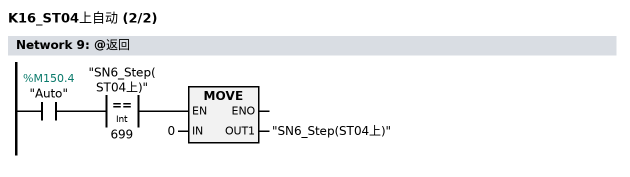
   RUNG wire#powerrail
      Contact( "Auto" )
      { S7_Templates := "SrcType := Int" } EQ_Contact(in1 := "SN6_Step(ST04上)", in2 := 699)
      Move(in := 0, out1 => "SN6_Step(ST04上)")
   END_RUNG
   // the same network as SCL:
   IF "Auto" AND ("SN6_Step(ST04上)" = 699) THEN "SN6_Step(ST04上)" := 0; END_IF;
END_REGION
END_FUNCTION_BLOCK

FUNCTION_BLOCK "K17_ST05上自动"   // FB17, LAD
{ S7_Optimized_Access := 'TRUE' }
VERSION : 0.1
// stored: AutoNumber false, IsIECCheckEnabled false, IsRetainMemResEnabled false, MemoryReserve 100, SetENOAutomatically false, UDAEnableTagReadback false
   VAR_TEMP   // added for the SCL form of the ladder/FBD networks
      _w1 : Bool;
   END_VAR
BEGIN

REGION Network 2: @搬出条件，SN7===ST05上工位
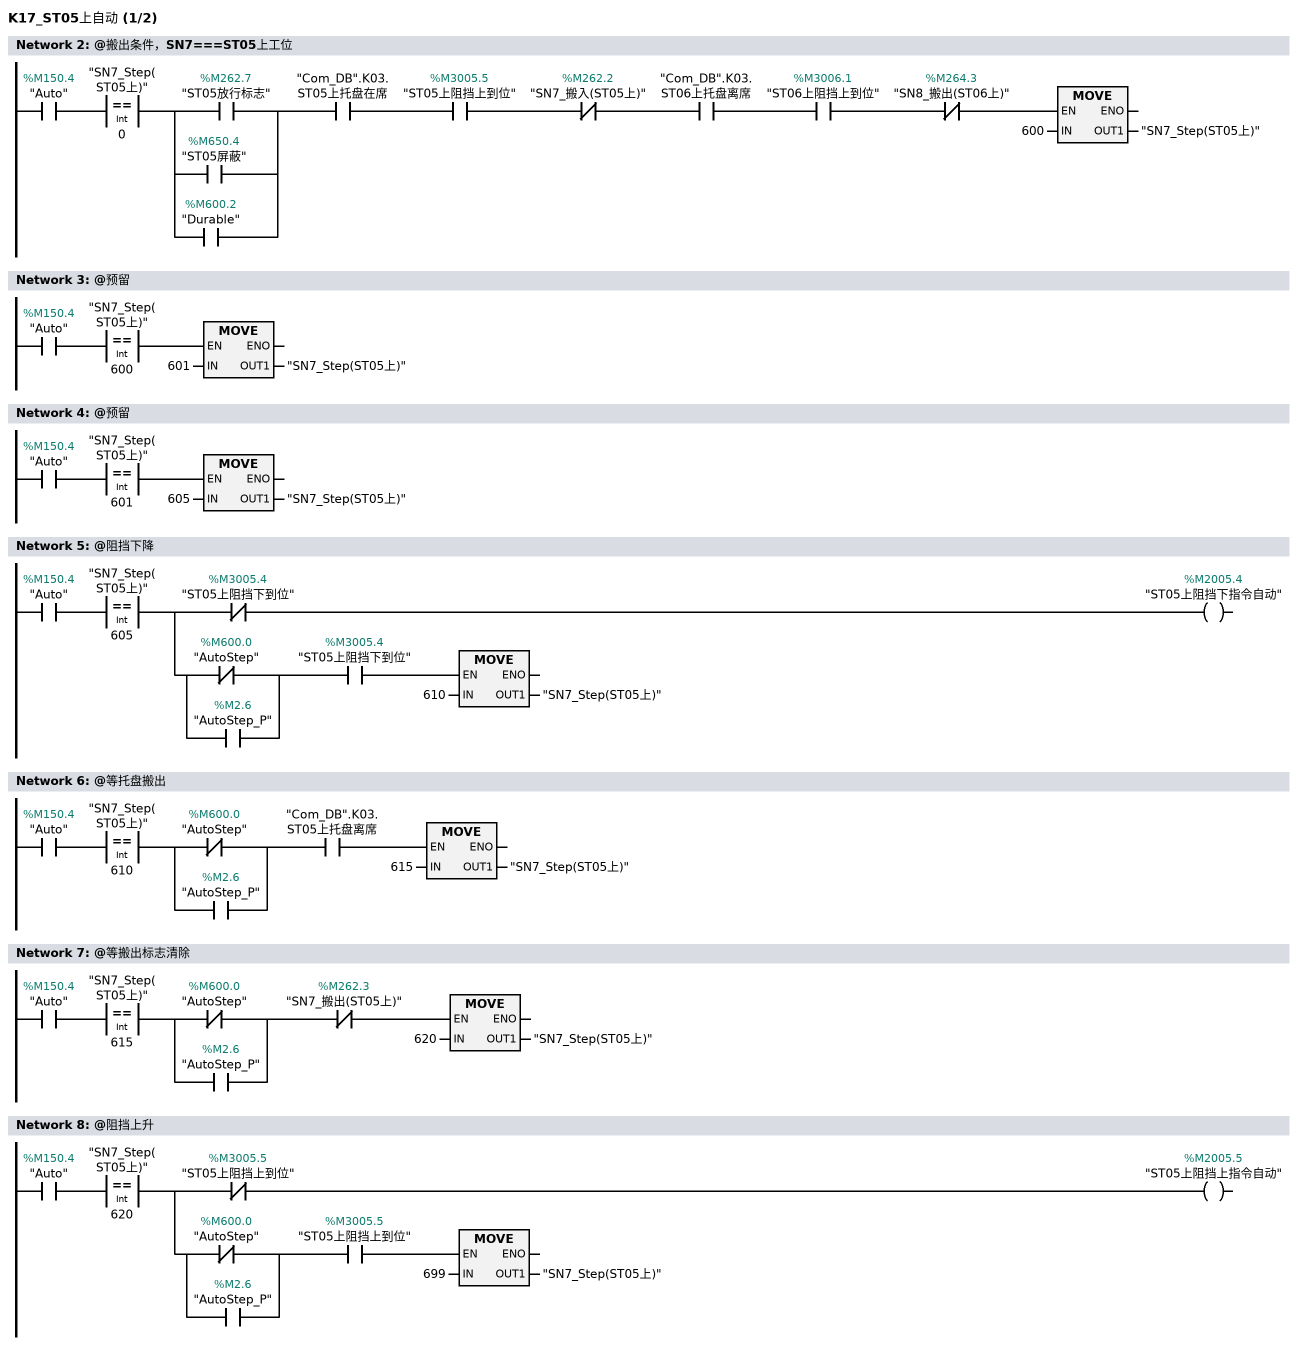
   RUNG wire#powerrail
      Contact( "Auto" )
      { S7_Templates := "SrcType := Int" } EQ_Contact(in1 := "SN7_Step(ST05上)", in2 := 0)
      wire#w1
      Contact( "ST05放行标志" )
      wire#w2
      Contact( "Com_DB".K03.ST05上托盘在席 )
      Contact( "ST05上阻挡上到位" )
      I_Contact( "SN7_搬入(ST05上)" )
      Contact( "Com_DB".K03.ST06上托盘离席 )
      Contact( "ST06上阻挡上到位" )
      I_Contact( "SN8_搬出(ST06上)" )
      Move(in := 600, out1 => "SN7_Step(ST05上)")
   END_RUNG
   RUNG wire#w1
      Contact( "ST05屏蔽" )
   END_RUNG wire#w2
   RUNG wire#w1
      Contact( "Durable" )
   END_RUNG wire#w2
   // the same network as SCL:
   IF "Auto" AND ("SN7_Step(ST05上)" = 0) AND ("ST05放行标志" OR "ST05屏蔽" OR "Durable") AND "Com_DB".K03.ST05上托盘在席 AND "ST05上阻挡上到位" AND NOT "SN7_搬入(ST05上)" AND "Com_DB".K03.ST06上托盘离席 AND "ST06上阻挡上到位" AND NOT "SN8_搬出(ST06上)" THEN
       "SN7_Step(ST05上)" := 600;
   END_IF;
END_REGION

REGION Network 3: @预留
   RUNG wire#powerrail
      Contact( "Auto" )
      { S7_Templates := "SrcType := Int" } EQ_Contact(in1 := "SN7_Step(ST05上)", in2 := 600)
      Move(in := 601, out1 => "SN7_Step(ST05上)")
   END_RUNG
   // the same network as SCL:
   IF "Auto" AND ("SN7_Step(ST05上)" = 600) THEN "SN7_Step(ST05上)" := 601; END_IF;
END_REGION

REGION Network 4: @预留
   RUNG wire#powerrail
      Contact( "Auto" )
      { S7_Templates := "SrcType := Int" } EQ_Contact(in1 := "SN7_Step(ST05上)", in2 := 601)
      Move(in := 605, out1 => "SN7_Step(ST05上)")
   END_RUNG
   // the same network as SCL:
   IF "Auto" AND ("SN7_Step(ST05上)" = 601) THEN "SN7_Step(ST05上)" := 605; END_IF;
END_REGION

REGION Network 5: @阻挡下降
   RUNG wire#powerrail
      Contact( "Auto" )
      { S7_Templates := "SrcType := Int" } EQ_Contact(in1 := "SN7_Step(ST05上)", in2 := 605)
      wire#w1
      I_Contact( "ST05上阻挡下到位" )
      Coil( "ST05上阻挡下指令自动" )
   END_RUNG
   RUNG wire#w1
      I_Contact( "AutoStep" )
      wire#w2
      Contact( "ST05上阻挡下到位" )
      Move(in := 610, out1 => "SN7_Step(ST05上)")
   END_RUNG
   RUNG wire#w1
      Contact( "AutoStep_P" )
   END_RUNG wire#w2
   // the same network as SCL:
   #_w1 := "Auto" AND ("SN7_Step(ST05上)" = 605);
   "ST05上阻挡下指令自动" := #_w1 AND NOT "ST05上阻挡下到位";
   IF #_w1 AND (NOT "AutoStep" OR "AutoStep_P") AND "ST05上阻挡下到位" THEN "SN7_Step(ST05上)" := 610; END_IF;
END_REGION

REGION Network 6: @等托盘搬出
   RUNG wire#powerrail
      Contact( "Auto" )
      { S7_Templates := "SrcType := Int" } EQ_Contact(in1 := "SN7_Step(ST05上)", in2 := 610)
      wire#w1
      I_Contact( "AutoStep" )
      wire#w2
      Contact( "Com_DB".K03.ST05上托盘离席 )
      Move(in := 615, out1 => "SN7_Step(ST05上)")
   END_RUNG
   RUNG wire#w1
      Contact( "AutoStep_P" )
   END_RUNG wire#w2
   // the same network as SCL:
   IF "Auto" AND ("SN7_Step(ST05上)" = 610) AND (NOT "AutoStep" OR "AutoStep_P") AND "Com_DB".K03.ST05上托盘离席 THEN
       "SN7_Step(ST05上)" := 615;
   END_IF;
END_REGION

REGION Network 7: @等搬出标志清除
   RUNG wire#powerrail
      Contact( "Auto" )
      { S7_Templates := "SrcType := Int" } EQ_Contact(in1 := "SN7_Step(ST05上)", in2 := 615)
      wire#w1
      I_Contact( "AutoStep" )
      wire#w2
      I_Contact( "SN7_搬出(ST05上)" )
      Move(in := 620, out1 => "SN7_Step(ST05上)")
   END_RUNG
   RUNG wire#w1
      Contact( "AutoStep_P" )
   END_RUNG wire#w2
   // the same network as SCL:
   IF "Auto" AND ("SN7_Step(ST05上)" = 615) AND (NOT "AutoStep" OR "AutoStep_P") AND NOT "SN7_搬出(ST05上)" THEN
       "SN7_Step(ST05上)" := 620;
   END_IF;
END_REGION

REGION Network 8: @阻挡上升
   RUNG wire#powerrail
      Contact( "Auto" )
      { S7_Templates := "SrcType := Int" } EQ_Contact(in1 := "SN7_Step(ST05上)", in2 := 620)
      wire#w1
      I_Contact( "ST05上阻挡上到位" )
      Coil( "ST05上阻挡上指令自动" )
   END_RUNG
   RUNG wire#w1
      I_Contact( "AutoStep" )
      wire#w2
      Contact( "ST05上阻挡上到位" )
      Move(in := 699, out1 => "SN7_Step(ST05上)")
   END_RUNG
   RUNG wire#w1
      Contact( "AutoStep_P" )
   END_RUNG wire#w2
   // the same network as SCL:
   #_w1 := "Auto" AND ("SN7_Step(ST05上)" = 620);
   "ST05上阻挡上指令自动" := #_w1 AND NOT "ST05上阻挡上到位";
   IF #_w1 AND (NOT "AutoStep" OR "AutoStep_P") AND "ST05上阻挡上到位" THEN "SN7_Step(ST05上)" := 699; END_IF;
END_REGION

REGION Network 9: @返回
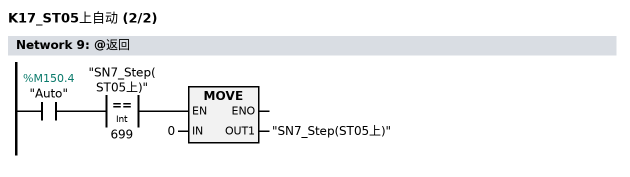
   RUNG wire#powerrail
      Contact( "Auto" )
      { S7_Templates := "SrcType := Int" } EQ_Contact(in1 := "SN7_Step(ST05上)", in2 := 699)
      Move(in := 0, out1 => "SN7_Step(ST05上)")
   END_RUNG
   // the same network as SCL:
   IF "Auto" AND ("SN7_Step(ST05上)" = 699) THEN "SN7_Step(ST05上)" := 0; END_IF;
END_REGION
END_FUNCTION_BLOCK

FUNCTION_BLOCK "K18_ST06上自动"   // FB18, LAD
{ S7_Optimized_Access := 'TRUE' }
VERSION : 0.1
// stored: AutoNumber false, IsIECCheckEnabled false, IsRetainMemResEnabled false, MemoryReserve 100, SetENOAutomatically false, UDAEnableTagReadback false
   VAR_TEMP   // added for the SCL form of the ladder/FBD networks
      _w1 : Bool;
   END_VAR
BEGIN

REGION Network 2: @搬出条件，SN8===ST06上工位
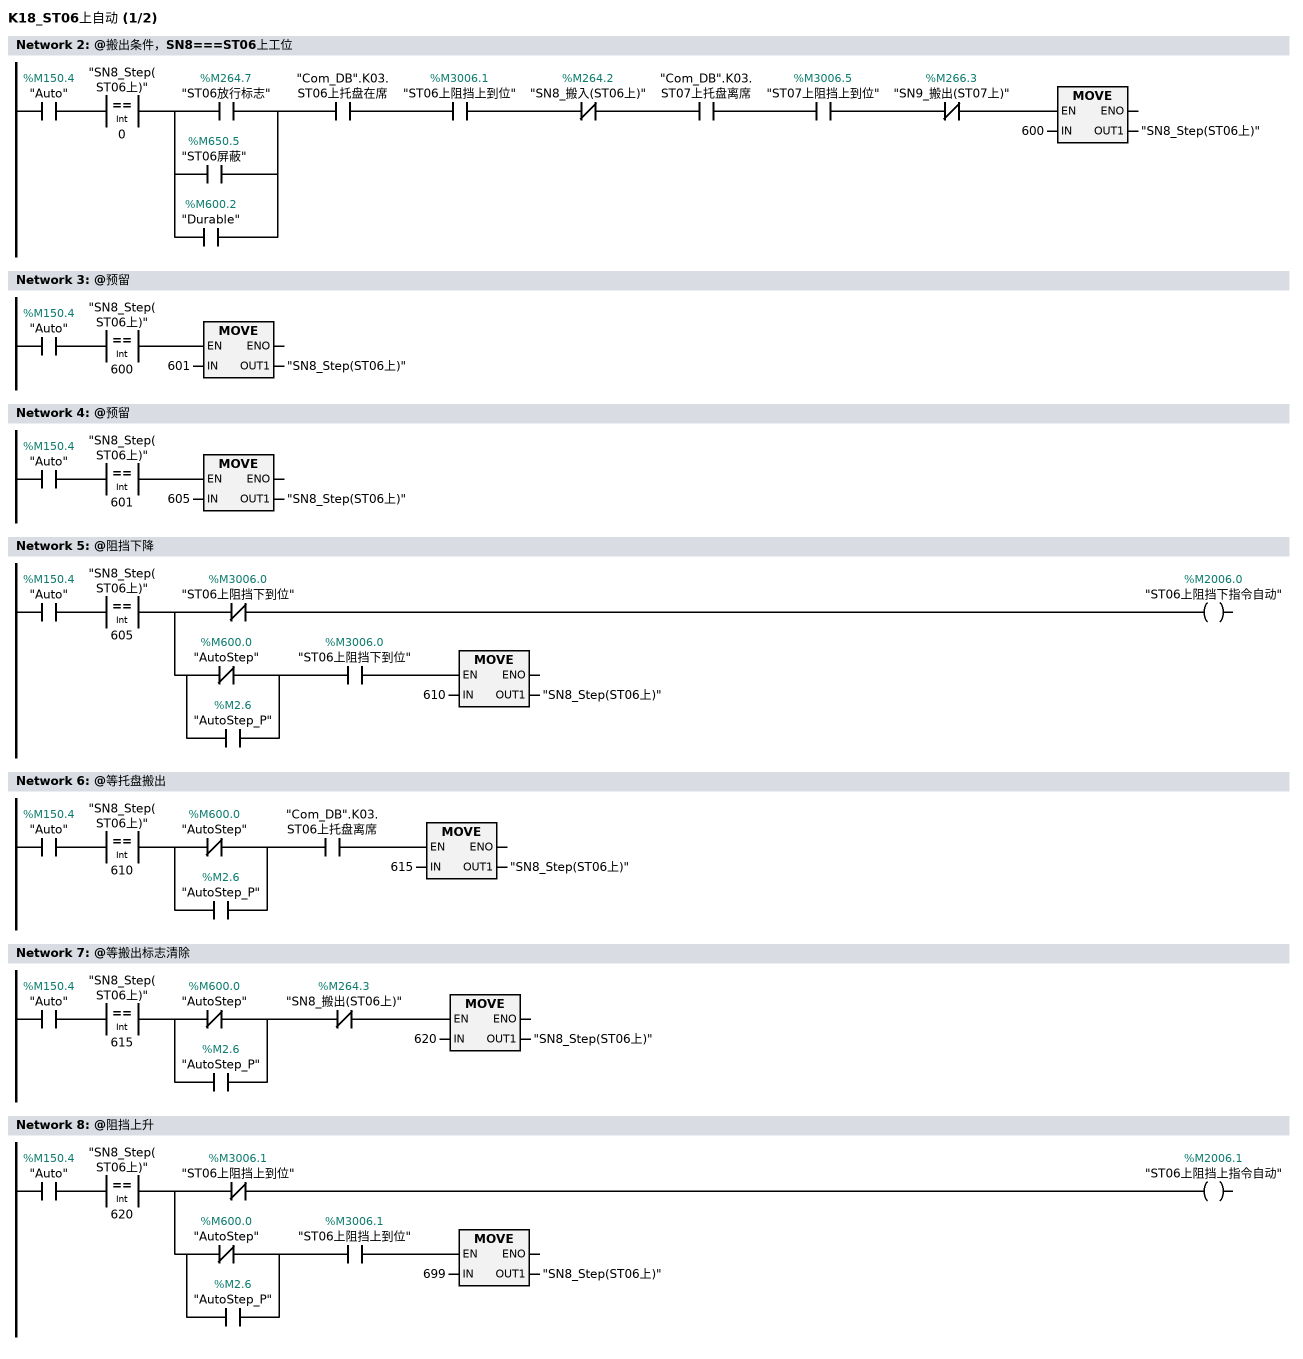
   RUNG wire#powerrail
      Contact( "Auto" )
      { S7_Templates := "SrcType := Int" } EQ_Contact(in1 := "SN8_Step(ST06上)", in2 := 0)
      wire#w1
      Contact( "ST06放行标志" )
      wire#w2
      Contact( "Com_DB".K03.ST06上托盘在席 )
      Contact( "ST06上阻挡上到位" )
      I_Contact( "SN8_搬入(ST06上)" )
      Contact( "Com_DB".K03.ST07上托盘离席 )
      Contact( "ST07上阻挡上到位" )
      I_Contact( "SN9_搬出(ST07上)" )
      Move(in := 600, out1 => "SN8_Step(ST06上)")
   END_RUNG
   RUNG wire#w1
      Contact( "ST06屏蔽" )
   END_RUNG wire#w2
   RUNG wire#w1
      Contact( "Durable" )
   END_RUNG wire#w2
   // the same network as SCL:
   IF "Auto" AND ("SN8_Step(ST06上)" = 0) AND ("ST06放行标志" OR "ST06屏蔽" OR "Durable") AND "Com_DB".K03.ST06上托盘在席 AND "ST06上阻挡上到位" AND NOT "SN8_搬入(ST06上)" AND "Com_DB".K03.ST07上托盘离席 AND "ST07上阻挡上到位" AND NOT "SN9_搬出(ST07上)" THEN
       "SN8_Step(ST06上)" := 600;
   END_IF;
END_REGION

REGION Network 3: @预留
   RUNG wire#powerrail
      Contact( "Auto" )
      { S7_Templates := "SrcType := Int" } EQ_Contact(in1 := "SN8_Step(ST06上)", in2 := 600)
      Move(in := 601, out1 => "SN8_Step(ST06上)")
   END_RUNG
   // the same network as SCL:
   IF "Auto" AND ("SN8_Step(ST06上)" = 600) THEN "SN8_Step(ST06上)" := 601; END_IF;
END_REGION

REGION Network 4: @预留
   RUNG wire#powerrail
      Contact( "Auto" )
      { S7_Templates := "SrcType := Int" } EQ_Contact(in1 := "SN8_Step(ST06上)", in2 := 601)
      Move(in := 605, out1 => "SN8_Step(ST06上)")
   END_RUNG
   // the same network as SCL:
   IF "Auto" AND ("SN8_Step(ST06上)" = 601) THEN "SN8_Step(ST06上)" := 605; END_IF;
END_REGION

REGION Network 5: @阻挡下降
   RUNG wire#powerrail
      Contact( "Auto" )
      { S7_Templates := "SrcType := Int" } EQ_Contact(in1 := "SN8_Step(ST06上)", in2 := 605)
      wire#w1
      I_Contact( "ST06上阻挡下到位" )
      Coil( "ST06上阻挡下指令自动" )
   END_RUNG
   RUNG wire#w1
      I_Contact( "AutoStep" )
      wire#w2
      Contact( "ST06上阻挡下到位" )
      Move(in := 610, out1 => "SN8_Step(ST06上)")
   END_RUNG
   RUNG wire#w1
      Contact( "AutoStep_P" )
   END_RUNG wire#w2
   // the same network as SCL:
   #_w1 := "Auto" AND ("SN8_Step(ST06上)" = 605);
   "ST06上阻挡下指令自动" := #_w1 AND NOT "ST06上阻挡下到位";
   IF #_w1 AND (NOT "AutoStep" OR "AutoStep_P") AND "ST06上阻挡下到位" THEN "SN8_Step(ST06上)" := 610; END_IF;
END_REGION

REGION Network 6: @等托盘搬出
   RUNG wire#powerrail
      Contact( "Auto" )
      { S7_Templates := "SrcType := Int" } EQ_Contact(in1 := "SN8_Step(ST06上)", in2 := 610)
      wire#w1
      I_Contact( "AutoStep" )
      wire#w2
      Contact( "Com_DB".K03.ST06上托盘离席 )
      Move(in := 615, out1 => "SN8_Step(ST06上)")
   END_RUNG
   RUNG wire#w1
      Contact( "AutoStep_P" )
   END_RUNG wire#w2
   // the same network as SCL:
   IF "Auto" AND ("SN8_Step(ST06上)" = 610) AND (NOT "AutoStep" OR "AutoStep_P") AND "Com_DB".K03.ST06上托盘离席 THEN
       "SN8_Step(ST06上)" := 615;
   END_IF;
END_REGION

REGION Network 7: @等搬出标志清除
   RUNG wire#powerrail
      Contact( "Auto" )
      { S7_Templates := "SrcType := Int" } EQ_Contact(in1 := "SN8_Step(ST06上)", in2 := 615)
      wire#w1
      I_Contact( "AutoStep" )
      wire#w2
      I_Contact( "SN8_搬出(ST06上)" )
      Move(in := 620, out1 => "SN8_Step(ST06上)")
   END_RUNG
   RUNG wire#w1
      Contact( "AutoStep_P" )
   END_RUNG wire#w2
   // the same network as SCL:
   IF "Auto" AND ("SN8_Step(ST06上)" = 615) AND (NOT "AutoStep" OR "AutoStep_P") AND NOT "SN8_搬出(ST06上)" THEN
       "SN8_Step(ST06上)" := 620;
   END_IF;
END_REGION

REGION Network 8: @阻挡上升
   RUNG wire#powerrail
      Contact( "Auto" )
      { S7_Templates := "SrcType := Int" } EQ_Contact(in1 := "SN8_Step(ST06上)", in2 := 620)
      wire#w1
      I_Contact( "ST06上阻挡上到位" )
      Coil( "ST06上阻挡上指令自动" )
   END_RUNG
   RUNG wire#w1
      I_Contact( "AutoStep" )
      wire#w2
      Contact( "ST06上阻挡上到位" )
      Move(in := 699, out1 => "SN8_Step(ST06上)")
   END_RUNG
   RUNG wire#w1
      Contact( "AutoStep_P" )
   END_RUNG wire#w2
   // the same network as SCL:
   #_w1 := "Auto" AND ("SN8_Step(ST06上)" = 620);
   "ST06上阻挡上指令自动" := #_w1 AND NOT "ST06上阻挡上到位";
   IF #_w1 AND (NOT "AutoStep" OR "AutoStep_P") AND "ST06上阻挡上到位" THEN "SN8_Step(ST06上)" := 699; END_IF;
END_REGION

REGION Network 9: @返回
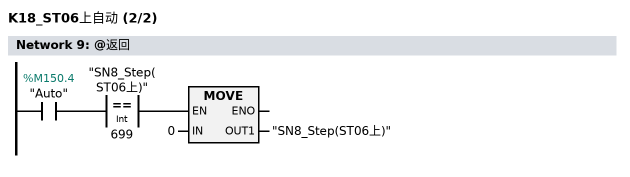
   RUNG wire#powerrail
      Contact( "Auto" )
      { S7_Templates := "SrcType := Int" } EQ_Contact(in1 := "SN8_Step(ST06上)", in2 := 699)
      Move(in := 0, out1 => "SN8_Step(ST06上)")
   END_RUNG
   // the same network as SCL:
   IF "Auto" AND ("SN8_Step(ST06上)" = 699) THEN "SN8_Step(ST06上)" := 0; END_IF;
END_REGION
END_FUNCTION_BLOCK

FUNCTION_BLOCK "K19_ST07上自动"   // FB19, LAD
{ S7_Optimized_Access := 'TRUE' }
VERSION : 0.1
// stored: AutoNumber false, IsIECCheckEnabled false, IsRetainMemResEnabled false, MemoryReserve 100, SetENOAutomatically false, UDAEnableTagReadback false
   VAR_TEMP   // added for the SCL form of the ladder/FBD networks
      _w1 : Bool;
   END_VAR
BEGIN

REGION Network 2: @搬出条件，SN9===ST07上工位
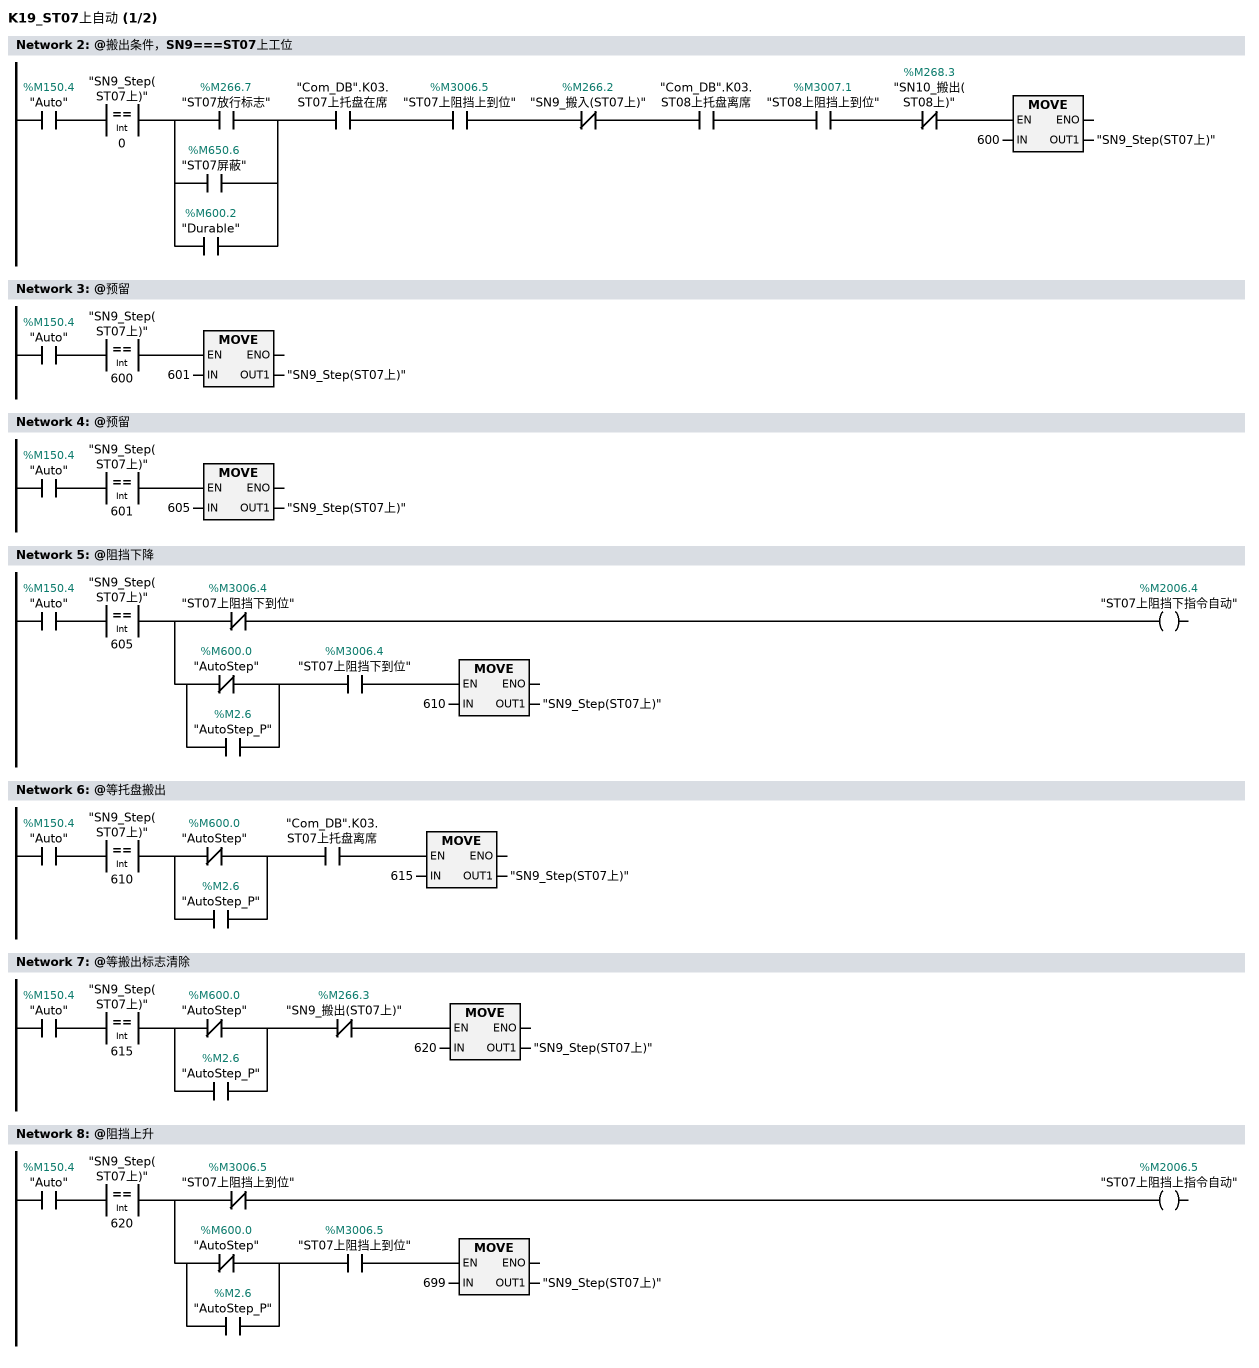
   RUNG wire#powerrail
      Contact( "Auto" )
      { S7_Templates := "SrcType := Int" } EQ_Contact(in1 := "SN9_Step(ST07上)", in2 := 0)
      wire#w1
      Contact( "ST07放行标志" )
      wire#w2
      Contact( "Com_DB".K03.ST07上托盘在席 )
      Contact( "ST07上阻挡上到位" )
      I_Contact( "SN9_搬入(ST07上)" )
      Contact( "Com_DB".K03.ST08上托盘离席 )
      Contact( "ST08上阻挡上到位" )
      I_Contact( "SN10_搬出(ST08上)" )
      Move(in := 600, out1 => "SN9_Step(ST07上)")
   END_RUNG
   RUNG wire#w1
      Contact( "ST07屏蔽" )
   END_RUNG wire#w2
   RUNG wire#w1
      Contact( "Durable" )
   END_RUNG wire#w2
   // the same network as SCL:
   IF "Auto" AND ("SN9_Step(ST07上)" = 0) AND ("ST07放行标志" OR "ST07屏蔽" OR "Durable") AND "Com_DB".K03.ST07上托盘在席 AND "ST07上阻挡上到位" AND NOT "SN9_搬入(ST07上)" AND "Com_DB".K03.ST08上托盘离席 AND "ST08上阻挡上到位" AND NOT "SN10_搬出(ST08上)" THEN
       "SN9_Step(ST07上)" := 600;
   END_IF;
END_REGION

REGION Network 3: @预留
   RUNG wire#powerrail
      Contact( "Auto" )
      { S7_Templates := "SrcType := Int" } EQ_Contact(in1 := "SN9_Step(ST07上)", in2 := 600)
      Move(in := 601, out1 => "SN9_Step(ST07上)")
   END_RUNG
   // the same network as SCL:
   IF "Auto" AND ("SN9_Step(ST07上)" = 600) THEN "SN9_Step(ST07上)" := 601; END_IF;
END_REGION

REGION Network 4: @预留
   RUNG wire#powerrail
      Contact( "Auto" )
      { S7_Templates := "SrcType := Int" } EQ_Contact(in1 := "SN9_Step(ST07上)", in2 := 601)
      Move(in := 605, out1 => "SN9_Step(ST07上)")
   END_RUNG
   // the same network as SCL:
   IF "Auto" AND ("SN9_Step(ST07上)" = 601) THEN "SN9_Step(ST07上)" := 605; END_IF;
END_REGION

REGION Network 5: @阻挡下降
   RUNG wire#powerrail
      Contact( "Auto" )
      { S7_Templates := "SrcType := Int" } EQ_Contact(in1 := "SN9_Step(ST07上)", in2 := 605)
      wire#w1
      I_Contact( "ST07上阻挡下到位" )
      Coil( "ST07上阻挡下指令自动" )
   END_RUNG
   RUNG wire#w1
      I_Contact( "AutoStep" )
      wire#w2
      Contact( "ST07上阻挡下到位" )
      Move(in := 610, out1 => "SN9_Step(ST07上)")
   END_RUNG
   RUNG wire#w1
      Contact( "AutoStep_P" )
   END_RUNG wire#w2
   // the same network as SCL:
   #_w1 := "Auto" AND ("SN9_Step(ST07上)" = 605);
   "ST07上阻挡下指令自动" := #_w1 AND NOT "ST07上阻挡下到位";
   IF #_w1 AND (NOT "AutoStep" OR "AutoStep_P") AND "ST07上阻挡下到位" THEN "SN9_Step(ST07上)" := 610; END_IF;
END_REGION

REGION Network 6: @等托盘搬出
   RUNG wire#powerrail
      Contact( "Auto" )
      { S7_Templates := "SrcType := Int" } EQ_Contact(in1 := "SN9_Step(ST07上)", in2 := 610)
      wire#w1
      I_Contact( "AutoStep" )
      wire#w2
      Contact( "Com_DB".K03.ST07上托盘离席 )
      Move(in := 615, out1 => "SN9_Step(ST07上)")
   END_RUNG
   RUNG wire#w1
      Contact( "AutoStep_P" )
   END_RUNG wire#w2
   // the same network as SCL:
   IF "Auto" AND ("SN9_Step(ST07上)" = 610) AND (NOT "AutoStep" OR "AutoStep_P") AND "Com_DB".K03.ST07上托盘离席 THEN
       "SN9_Step(ST07上)" := 615;
   END_IF;
END_REGION

REGION Network 7: @等搬出标志清除
   RUNG wire#powerrail
      Contact( "Auto" )
      { S7_Templates := "SrcType := Int" } EQ_Contact(in1 := "SN9_Step(ST07上)", in2 := 615)
      wire#w1
      I_Contact( "AutoStep" )
      wire#w2
      I_Contact( "SN9_搬出(ST07上)" )
      Move(in := 620, out1 => "SN9_Step(ST07上)")
   END_RUNG
   RUNG wire#w1
      Contact( "AutoStep_P" )
   END_RUNG wire#w2
   // the same network as SCL:
   IF "Auto" AND ("SN9_Step(ST07上)" = 615) AND (NOT "AutoStep" OR "AutoStep_P") AND NOT "SN9_搬出(ST07上)" THEN
       "SN9_Step(ST07上)" := 620;
   END_IF;
END_REGION

REGION Network 8: @阻挡上升
   RUNG wire#powerrail
      Contact( "Auto" )
      { S7_Templates := "SrcType := Int" } EQ_Contact(in1 := "SN9_Step(ST07上)", in2 := 620)
      wire#w1
      I_Contact( "ST07上阻挡上到位" )
      Coil( "ST07上阻挡上指令自动" )
   END_RUNG
   RUNG wire#w1
      I_Contact( "AutoStep" )
      wire#w2
      Contact( "ST07上阻挡上到位" )
      Move(in := 699, out1 => "SN9_Step(ST07上)")
   END_RUNG
   RUNG wire#w1
      Contact( "AutoStep_P" )
   END_RUNG wire#w2
   // the same network as SCL:
   #_w1 := "Auto" AND ("SN9_Step(ST07上)" = 620);
   "ST07上阻挡上指令自动" := #_w1 AND NOT "ST07上阻挡上到位";
   IF #_w1 AND (NOT "AutoStep" OR "AutoStep_P") AND "ST07上阻挡上到位" THEN "SN9_Step(ST07上)" := 699; END_IF;
END_REGION

REGION Network 9: @返回
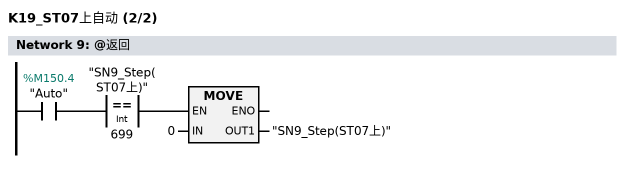
   RUNG wire#powerrail
      Contact( "Auto" )
      { S7_Templates := "SrcType := Int" } EQ_Contact(in1 := "SN9_Step(ST07上)", in2 := 699)
      Move(in := 0, out1 => "SN9_Step(ST07上)")
   END_RUNG
   // the same network as SCL:
   IF "Auto" AND ("SN9_Step(ST07上)" = 699) THEN "SN9_Step(ST07上)" := 0; END_IF;
END_REGION
END_FUNCTION_BLOCK

FUNCTION_BLOCK "K20_ST08上自动"   // FB20, LAD
{ S7_Optimized_Access := 'TRUE' }
VERSION : 0.1
// stored: AutoNumber false, IsIECCheckEnabled false, IsRetainMemResEnabled false, MemoryReserve 100, SetENOAutomatically false, UDAEnableTagReadback false
   VAR_TEMP   // added for the SCL form of the ladder/FBD networks
      _w1 : Bool;
   END_VAR
BEGIN

REGION Network 2: @搬出条件，SN10===ST08上工位
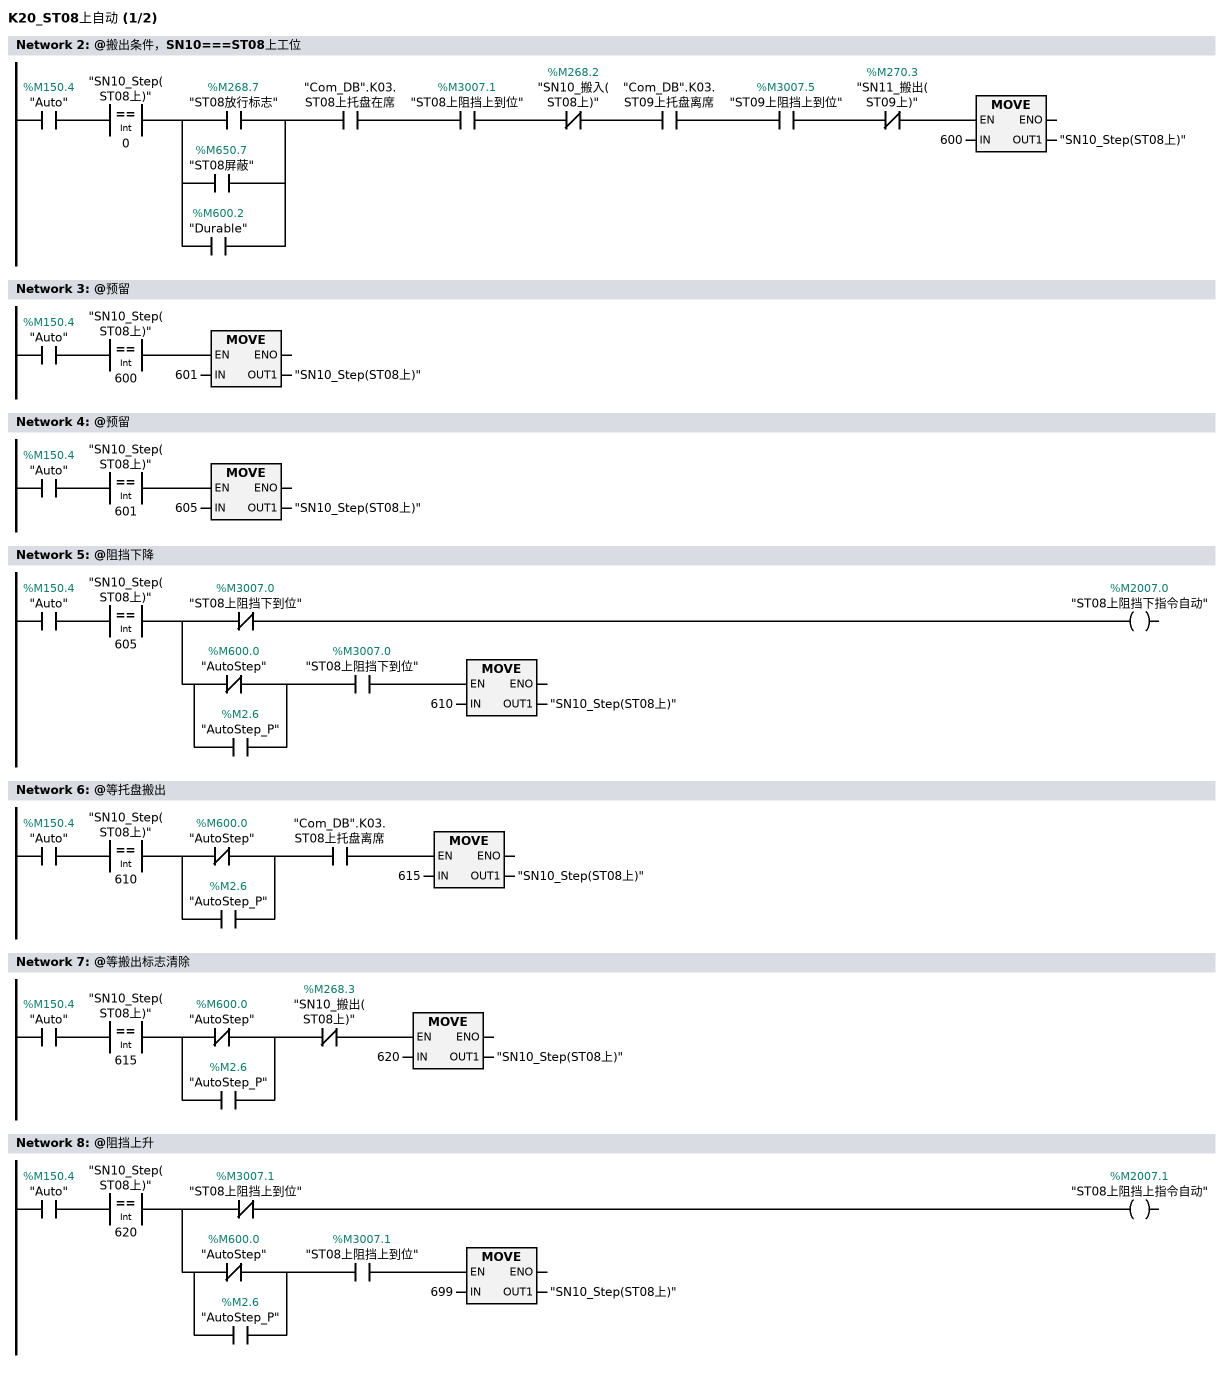
   RUNG wire#powerrail
      Contact( "Auto" )
      { S7_Templates := "SrcType := Int" } EQ_Contact(in1 := "SN10_Step(ST08上)", in2 := 0)
      wire#w1
      Contact( "ST08放行标志" )
      wire#w2
      Contact( "Com_DB".K03.ST08上托盘在席 )
      Contact( "ST08上阻挡上到位" )
      I_Contact( "SN10_搬入(ST08上)" )
      Contact( "Com_DB".K03.ST09上托盘离席 )
      Contact( "ST09上阻挡上到位" )
      I_Contact( "SN11_搬出(ST09上)" )
      Move(in := 600, out1 => "SN10_Step(ST08上)")
   END_RUNG
   RUNG wire#w1
      Contact( "ST08屏蔽" )
   END_RUNG wire#w2
   RUNG wire#w1
      Contact( "Durable" )
   END_RUNG wire#w2
   // the same network as SCL:
   IF "Auto" AND ("SN10_Step(ST08上)" = 0) AND ("ST08放行标志" OR "ST08屏蔽" OR "Durable") AND "Com_DB".K03.ST08上托盘在席 AND "ST08上阻挡上到位" AND NOT "SN10_搬入(ST08上)" AND "Com_DB".K03.ST09上托盘离席 AND "ST09上阻挡上到位" AND NOT "SN11_搬出(ST09上)" THEN
       "SN10_Step(ST08上)" := 600;
   END_IF;
END_REGION

REGION Network 3: @预留
   RUNG wire#powerrail
      Contact( "Auto" )
      { S7_Templates := "SrcType := Int" } EQ_Contact(in1 := "SN10_Step(ST08上)", in2 := 600)
      Move(in := 601, out1 => "SN10_Step(ST08上)")
   END_RUNG
   // the same network as SCL:
   IF "Auto" AND ("SN10_Step(ST08上)" = 600) THEN "SN10_Step(ST08上)" := 601; END_IF;
END_REGION

REGION Network 4: @预留
   RUNG wire#powerrail
      Contact( "Auto" )
      { S7_Templates := "SrcType := Int" } EQ_Contact(in1 := "SN10_Step(ST08上)", in2 := 601)
      Move(in := 605, out1 => "SN10_Step(ST08上)")
   END_RUNG
   // the same network as SCL:
   IF "Auto" AND ("SN10_Step(ST08上)" = 601) THEN "SN10_Step(ST08上)" := 605; END_IF;
END_REGION

REGION Network 5: @阻挡下降
   RUNG wire#powerrail
      Contact( "Auto" )
      { S7_Templates := "SrcType := Int" } EQ_Contact(in1 := "SN10_Step(ST08上)", in2 := 605)
      wire#w1
      I_Contact( "ST08上阻挡下到位" )
      Coil( "ST08上阻挡下指令自动" )
   END_RUNG
   RUNG wire#w1
      I_Contact( "AutoStep" )
      wire#w2
      Contact( "ST08上阻挡下到位" )
      Move(in := 610, out1 => "SN10_Step(ST08上)")
   END_RUNG
   RUNG wire#w1
      Contact( "AutoStep_P" )
   END_RUNG wire#w2
   // the same network as SCL:
   #_w1 := "Auto" AND ("SN10_Step(ST08上)" = 605);
   "ST08上阻挡下指令自动" := #_w1 AND NOT "ST08上阻挡下到位";
   IF #_w1 AND (NOT "AutoStep" OR "AutoStep_P") AND "ST08上阻挡下到位" THEN "SN10_Step(ST08上)" := 610; END_IF;
END_REGION

REGION Network 6: @等托盘搬出
   RUNG wire#powerrail
      Contact( "Auto" )
      { S7_Templates := "SrcType := Int" } EQ_Contact(in1 := "SN10_Step(ST08上)", in2 := 610)
      wire#w1
      I_Contact( "AutoStep" )
      wire#w2
      Contact( "Com_DB".K03.ST08上托盘离席 )
      Move(in := 615, out1 => "SN10_Step(ST08上)")
   END_RUNG
   RUNG wire#w1
      Contact( "AutoStep_P" )
   END_RUNG wire#w2
   // the same network as SCL:
   IF "Auto" AND ("SN10_Step(ST08上)" = 610) AND (NOT "AutoStep" OR "AutoStep_P") AND "Com_DB".K03.ST08上托盘离席 THEN
       "SN10_Step(ST08上)" := 615;
   END_IF;
END_REGION

REGION Network 7: @等搬出标志清除
   RUNG wire#powerrail
      Contact( "Auto" )
      { S7_Templates := "SrcType := Int" } EQ_Contact(in1 := "SN10_Step(ST08上)", in2 := 615)
      wire#w1
      I_Contact( "AutoStep" )
      wire#w2
      I_Contact( "SN10_搬出(ST08上)" )
      Move(in := 620, out1 => "SN10_Step(ST08上)")
   END_RUNG
   RUNG wire#w1
      Contact( "AutoStep_P" )
   END_RUNG wire#w2
   // the same network as SCL:
   IF "Auto" AND ("SN10_Step(ST08上)" = 615) AND (NOT "AutoStep" OR "AutoStep_P") AND NOT "SN10_搬出(ST08上)" THEN
       "SN10_Step(ST08上)" := 620;
   END_IF;
END_REGION

REGION Network 8: @阻挡上升
   RUNG wire#powerrail
      Contact( "Auto" )
      { S7_Templates := "SrcType := Int" } EQ_Contact(in1 := "SN10_Step(ST08上)", in2 := 620)
      wire#w1
      I_Contact( "ST08上阻挡上到位" )
      Coil( "ST08上阻挡上指令自动" )
   END_RUNG
   RUNG wire#w1
      I_Contact( "AutoStep" )
      wire#w2
      Contact( "ST08上阻挡上到位" )
      Move(in := 699, out1 => "SN10_Step(ST08上)")
   END_RUNG
   RUNG wire#w1
      Contact( "AutoStep_P" )
   END_RUNG wire#w2
   // the same network as SCL:
   #_w1 := "Auto" AND ("SN10_Step(ST08上)" = 620);
   "ST08上阻挡上指令自动" := #_w1 AND NOT "ST08上阻挡上到位";
   IF #_w1 AND (NOT "AutoStep" OR "AutoStep_P") AND "ST08上阻挡上到位" THEN "SN10_Step(ST08上)" := 699; END_IF;
END_REGION

REGION Network 9: @返回
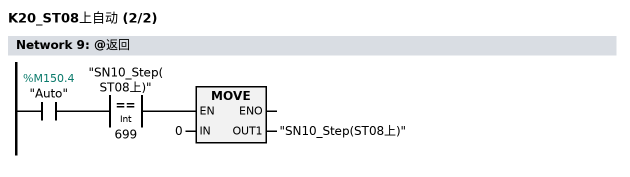
   RUNG wire#powerrail
      Contact( "Auto" )
      { S7_Templates := "SrcType := Int" } EQ_Contact(in1 := "SN10_Step(ST08上)", in2 := 699)
      Move(in := 0, out1 => "SN10_Step(ST08上)")
   END_RUNG
   // the same network as SCL:
   IF "Auto" AND ("SN10_Step(ST08上)" = 699) THEN "SN10_Step(ST08上)" := 0; END_IF;
END_REGION
END_FUNCTION_BLOCK

FUNCTION_BLOCK "K21_ST09上自动"   // FB21, LAD
{ S7_Optimized_Access := 'TRUE' }
VERSION : 0.1
// stored: AutoNumber false, IsIECCheckEnabled false, IsRetainMemResEnabled false, MemoryReserve 100, SetENOAutomatically false, UDAEnableTagReadback false
   VAR_TEMP   // added for the SCL form of the ladder/FBD networks
      _w1 : Bool;
   END_VAR
BEGIN

REGION Network 2: @搬出条件，SN11===ST09上工位
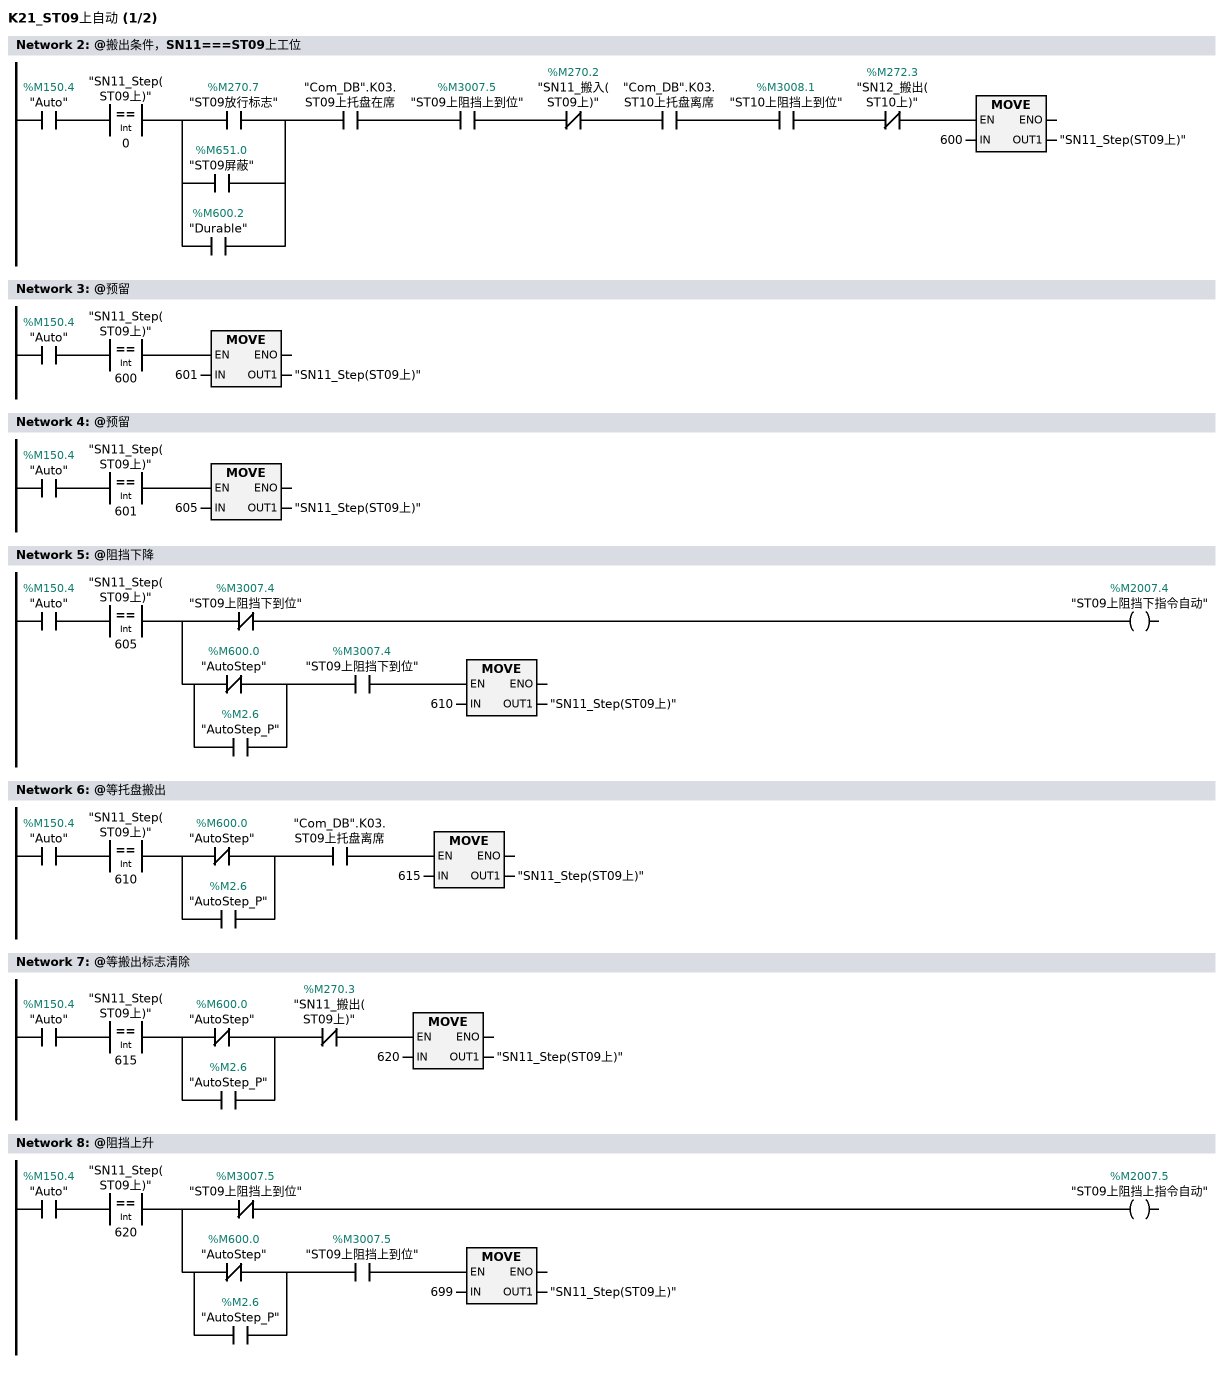
   RUNG wire#powerrail
      Contact( "Auto" )
      { S7_Templates := "SrcType := Int" } EQ_Contact(in1 := "SN11_Step(ST09上)", in2 := 0)
      wire#w1
      Contact( "ST09放行标志" )
      wire#w2
      Contact( "Com_DB".K03.ST09上托盘在席 )
      Contact( "ST09上阻挡上到位" )
      I_Contact( "SN11_搬入(ST09上)" )
      Contact( "Com_DB".K03.ST10上托盘离席 )
      Contact( "ST10上阻挡上到位" )
      I_Contact( "SN12_搬出(ST10上)" )
      Move(in := 600, out1 => "SN11_Step(ST09上)")
   END_RUNG
   RUNG wire#w1
      Contact( "ST09屏蔽" )
   END_RUNG wire#w2
   RUNG wire#w1
      Contact( "Durable" )
   END_RUNG wire#w2
   // the same network as SCL:
   IF "Auto" AND ("SN11_Step(ST09上)" = 0) AND ("ST09放行标志" OR "ST09屏蔽" OR "Durable") AND "Com_DB".K03.ST09上托盘在席 AND "ST09上阻挡上到位" AND NOT "SN11_搬入(ST09上)" AND "Com_DB".K03.ST10上托盘离席 AND "ST10上阻挡上到位" AND NOT "SN12_搬出(ST10上)" THEN
       "SN11_Step(ST09上)" := 600;
   END_IF;
END_REGION

REGION Network 3: @预留
   RUNG wire#powerrail
      Contact( "Auto" )
      { S7_Templates := "SrcType := Int" } EQ_Contact(in1 := "SN11_Step(ST09上)", in2 := 600)
      Move(in := 601, out1 => "SN11_Step(ST09上)")
   END_RUNG
   // the same network as SCL:
   IF "Auto" AND ("SN11_Step(ST09上)" = 600) THEN "SN11_Step(ST09上)" := 601; END_IF;
END_REGION

REGION Network 4: @预留
   RUNG wire#powerrail
      Contact( "Auto" )
      { S7_Templates := "SrcType := Int" } EQ_Contact(in1 := "SN11_Step(ST09上)", in2 := 601)
      Move(in := 605, out1 => "SN11_Step(ST09上)")
   END_RUNG
   // the same network as SCL:
   IF "Auto" AND ("SN11_Step(ST09上)" = 601) THEN "SN11_Step(ST09上)" := 605; END_IF;
END_REGION

REGION Network 5: @阻挡下降
   RUNG wire#powerrail
      Contact( "Auto" )
      { S7_Templates := "SrcType := Int" } EQ_Contact(in1 := "SN11_Step(ST09上)", in2 := 605)
      wire#w1
      I_Contact( "ST09上阻挡下到位" )
      Coil( "ST09上阻挡下指令自动" )
   END_RUNG
   RUNG wire#w1
      I_Contact( "AutoStep" )
      wire#w2
      Contact( "ST09上阻挡下到位" )
      Move(in := 610, out1 => "SN11_Step(ST09上)")
   END_RUNG
   RUNG wire#w1
      Contact( "AutoStep_P" )
   END_RUNG wire#w2
   // the same network as SCL:
   #_w1 := "Auto" AND ("SN11_Step(ST09上)" = 605);
   "ST09上阻挡下指令自动" := #_w1 AND NOT "ST09上阻挡下到位";
   IF #_w1 AND (NOT "AutoStep" OR "AutoStep_P") AND "ST09上阻挡下到位" THEN "SN11_Step(ST09上)" := 610; END_IF;
END_REGION

REGION Network 6: @等托盘搬出
   RUNG wire#powerrail
      Contact( "Auto" )
      { S7_Templates := "SrcType := Int" } EQ_Contact(in1 := "SN11_Step(ST09上)", in2 := 610)
      wire#w1
      I_Contact( "AutoStep" )
      wire#w2
      Contact( "Com_DB".K03.ST09上托盘离席 )
      Move(in := 615, out1 => "SN11_Step(ST09上)")
   END_RUNG
   RUNG wire#w1
      Contact( "AutoStep_P" )
   END_RUNG wire#w2
   // the same network as SCL:
   IF "Auto" AND ("SN11_Step(ST09上)" = 610) AND (NOT "AutoStep" OR "AutoStep_P") AND "Com_DB".K03.ST09上托盘离席 THEN
       "SN11_Step(ST09上)" := 615;
   END_IF;
END_REGION

REGION Network 7: @等搬出标志清除
   RUNG wire#powerrail
      Contact( "Auto" )
      { S7_Templates := "SrcType := Int" } EQ_Contact(in1 := "SN11_Step(ST09上)", in2 := 615)
      wire#w1
      I_Contact( "AutoStep" )
      wire#w2
      I_Contact( "SN11_搬出(ST09上)" )
      Move(in := 620, out1 => "SN11_Step(ST09上)")
   END_RUNG
   RUNG wire#w1
      Contact( "AutoStep_P" )
   END_RUNG wire#w2
   // the same network as SCL:
   IF "Auto" AND ("SN11_Step(ST09上)" = 615) AND (NOT "AutoStep" OR "AutoStep_P") AND NOT "SN11_搬出(ST09上)" THEN
       "SN11_Step(ST09上)" := 620;
   END_IF;
END_REGION

REGION Network 8: @阻挡上升
   RUNG wire#powerrail
      Contact( "Auto" )
      { S7_Templates := "SrcType := Int" } EQ_Contact(in1 := "SN11_Step(ST09上)", in2 := 620)
      wire#w1
      I_Contact( "ST09上阻挡上到位" )
      Coil( "ST09上阻挡上指令自动" )
   END_RUNG
   RUNG wire#w1
      I_Contact( "AutoStep" )
      wire#w2
      Contact( "ST09上阻挡上到位" )
      Move(in := 699, out1 => "SN11_Step(ST09上)")
   END_RUNG
   RUNG wire#w1
      Contact( "AutoStep_P" )
   END_RUNG wire#w2
   // the same network as SCL:
   #_w1 := "Auto" AND ("SN11_Step(ST09上)" = 620);
   "ST09上阻挡上指令自动" := #_w1 AND NOT "ST09上阻挡上到位";
   IF #_w1 AND (NOT "AutoStep" OR "AutoStep_P") AND "ST09上阻挡上到位" THEN "SN11_Step(ST09上)" := 699; END_IF;
END_REGION

REGION Network 9: @返回
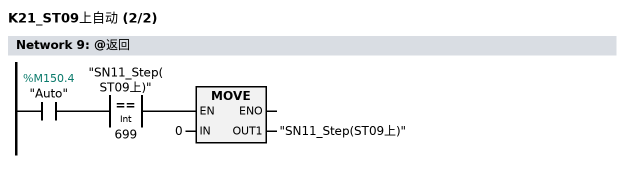
   RUNG wire#powerrail
      Contact( "Auto" )
      { S7_Templates := "SrcType := Int" } EQ_Contact(in1 := "SN11_Step(ST09上)", in2 := 699)
      Move(in := 0, out1 => "SN11_Step(ST09上)")
   END_RUNG
   // the same network as SCL:
   IF "Auto" AND ("SN11_Step(ST09上)" = 699) THEN "SN11_Step(ST09上)" := 0; END_IF;
END_REGION
END_FUNCTION_BLOCK

FUNCTION_BLOCK "K22_ST10上自动"   // FB22, LAD
{ S7_Optimized_Access := 'TRUE' }
VERSION : 0.1
// stored: AutoNumber false, IsIECCheckEnabled false, IsRetainMemResEnabled false, MemoryReserve 100, SetENOAutomatically false, UDAEnableTagReadback false
   VAR_TEMP   // added for the SCL form of the ladder/FBD networks
      _w1 : Bool;
   END_VAR
BEGIN

REGION Network 2: @搬出条件，SN12===ST10上工位
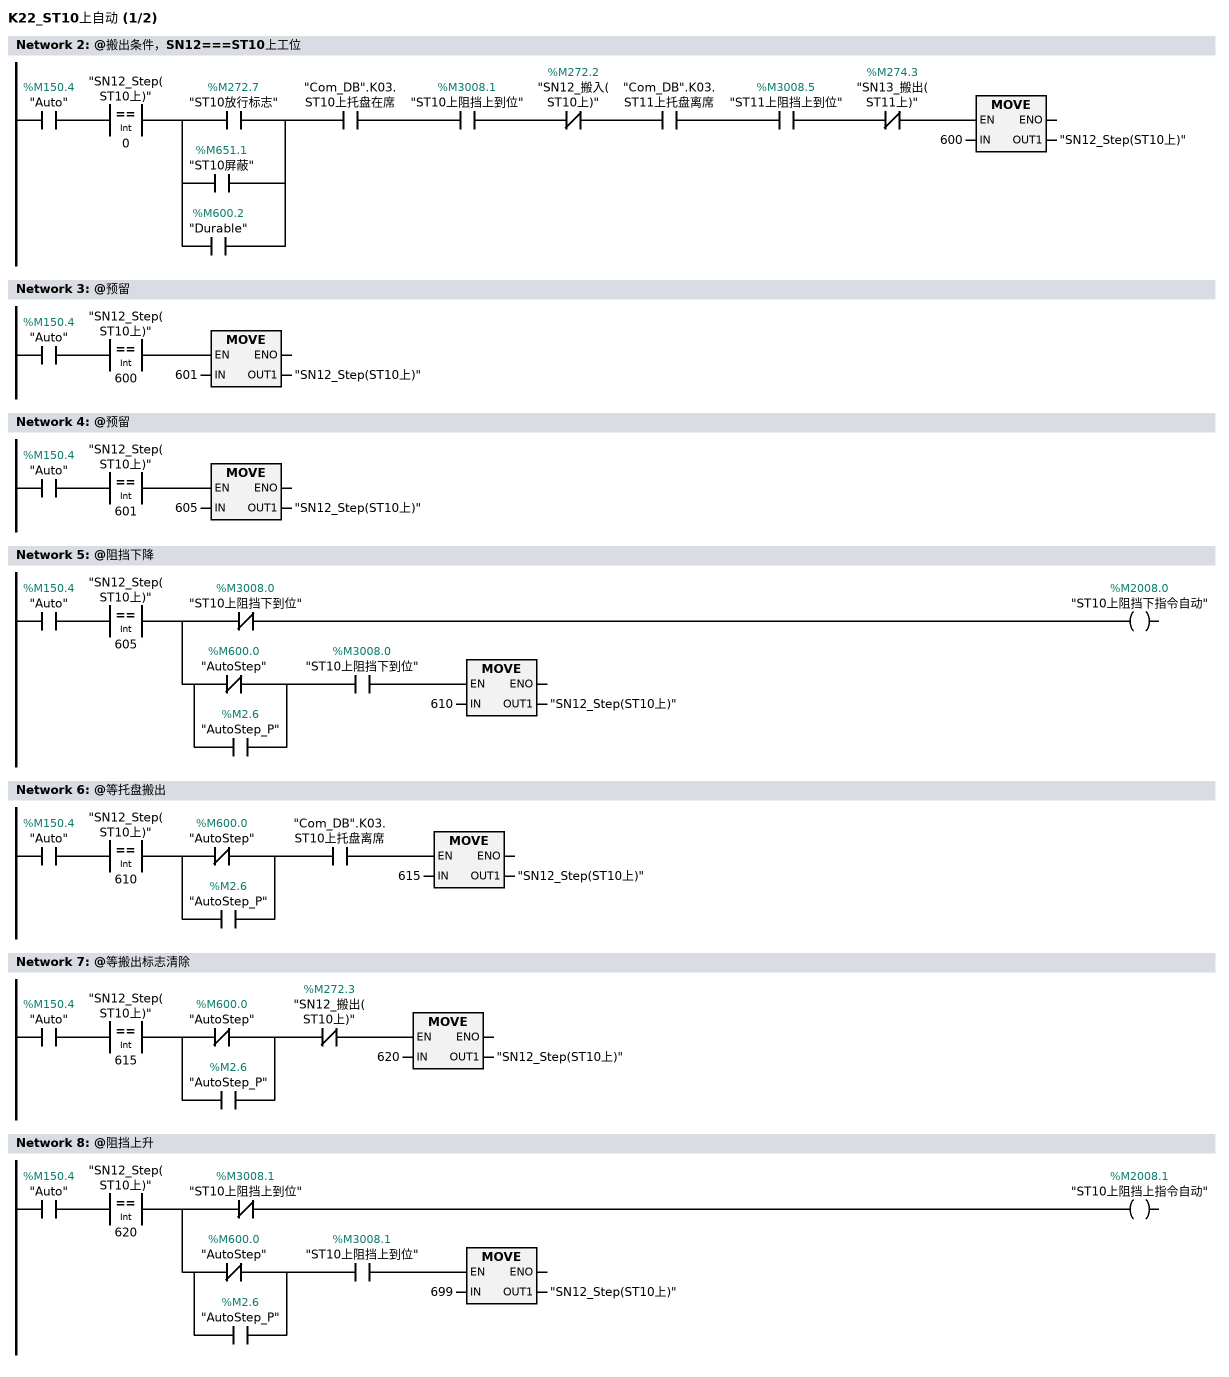
   RUNG wire#powerrail
      Contact( "Auto" )
      { S7_Templates := "SrcType := Int" } EQ_Contact(in1 := "SN12_Step(ST10上)", in2 := 0)
      wire#w1
      Contact( "ST10放行标志" )
      wire#w2
      Contact( "Com_DB".K03.ST10上托盘在席 )
      Contact( "ST10上阻挡上到位" )
      I_Contact( "SN12_搬入(ST10上)" )
      Contact( "Com_DB".K03.ST11上托盘离席 )
      Contact( "ST11上阻挡上到位" )
      I_Contact( "SN13_搬出(ST11上)" )
      Move(in := 600, out1 => "SN12_Step(ST10上)")
   END_RUNG
   RUNG wire#w1
      Contact( "ST10屏蔽" )
   END_RUNG wire#w2
   RUNG wire#w1
      Contact( "Durable" )
   END_RUNG wire#w2
   // the same network as SCL:
   IF "Auto" AND ("SN12_Step(ST10上)" = 0) AND ("ST10放行标志" OR "ST10屏蔽" OR "Durable") AND "Com_DB".K03.ST10上托盘在席 AND "ST10上阻挡上到位" AND NOT "SN12_搬入(ST10上)" AND "Com_DB".K03.ST11上托盘离席 AND "ST11上阻挡上到位" AND NOT "SN13_搬出(ST11上)" THEN
       "SN12_Step(ST10上)" := 600;
   END_IF;
END_REGION

REGION Network 3: @预留
   RUNG wire#powerrail
      Contact( "Auto" )
      { S7_Templates := "SrcType := Int" } EQ_Contact(in1 := "SN12_Step(ST10上)", in2 := 600)
      Move(in := 601, out1 => "SN12_Step(ST10上)")
   END_RUNG
   // the same network as SCL:
   IF "Auto" AND ("SN12_Step(ST10上)" = 600) THEN "SN12_Step(ST10上)" := 601; END_IF;
END_REGION

REGION Network 4: @预留
   RUNG wire#powerrail
      Contact( "Auto" )
      { S7_Templates := "SrcType := Int" } EQ_Contact(in1 := "SN12_Step(ST10上)", in2 := 601)
      Move(in := 605, out1 => "SN12_Step(ST10上)")
   END_RUNG
   // the same network as SCL:
   IF "Auto" AND ("SN12_Step(ST10上)" = 601) THEN "SN12_Step(ST10上)" := 605; END_IF;
END_REGION

REGION Network 5: @阻挡下降
   RUNG wire#powerrail
      Contact( "Auto" )
      { S7_Templates := "SrcType := Int" } EQ_Contact(in1 := "SN12_Step(ST10上)", in2 := 605)
      wire#w1
      I_Contact( "ST10上阻挡下到位" )
      Coil( "ST10上阻挡下指令自动" )
   END_RUNG
   RUNG wire#w1
      I_Contact( "AutoStep" )
      wire#w2
      Contact( "ST10上阻挡下到位" )
      Move(in := 610, out1 => "SN12_Step(ST10上)")
   END_RUNG
   RUNG wire#w1
      Contact( "AutoStep_P" )
   END_RUNG wire#w2
   // the same network as SCL:
   #_w1 := "Auto" AND ("SN12_Step(ST10上)" = 605);
   "ST10上阻挡下指令自动" := #_w1 AND NOT "ST10上阻挡下到位";
   IF #_w1 AND (NOT "AutoStep" OR "AutoStep_P") AND "ST10上阻挡下到位" THEN "SN12_Step(ST10上)" := 610; END_IF;
END_REGION

REGION Network 6: @等托盘搬出
   RUNG wire#powerrail
      Contact( "Auto" )
      { S7_Templates := "SrcType := Int" } EQ_Contact(in1 := "SN12_Step(ST10上)", in2 := 610)
      wire#w1
      I_Contact( "AutoStep" )
      wire#w2
      Contact( "Com_DB".K03.ST10上托盘离席 )
      Move(in := 615, out1 => "SN12_Step(ST10上)")
   END_RUNG
   RUNG wire#w1
      Contact( "AutoStep_P" )
   END_RUNG wire#w2
   // the same network as SCL:
   IF "Auto" AND ("SN12_Step(ST10上)" = 610) AND (NOT "AutoStep" OR "AutoStep_P") AND "Com_DB".K03.ST10上托盘离席 THEN
       "SN12_Step(ST10上)" := 615;
   END_IF;
END_REGION

REGION Network 7: @等搬出标志清除
   RUNG wire#powerrail
      Contact( "Auto" )
      { S7_Templates := "SrcType := Int" } EQ_Contact(in1 := "SN12_Step(ST10上)", in2 := 615)
      wire#w1
      I_Contact( "AutoStep" )
      wire#w2
      I_Contact( "SN12_搬出(ST10上)" )
      Move(in := 620, out1 => "SN12_Step(ST10上)")
   END_RUNG
   RUNG wire#w1
      Contact( "AutoStep_P" )
   END_RUNG wire#w2
   // the same network as SCL:
   IF "Auto" AND ("SN12_Step(ST10上)" = 615) AND (NOT "AutoStep" OR "AutoStep_P") AND NOT "SN12_搬出(ST10上)" THEN
       "SN12_Step(ST10上)" := 620;
   END_IF;
END_REGION

REGION Network 8: @阻挡上升
   RUNG wire#powerrail
      Contact( "Auto" )
      { S7_Templates := "SrcType := Int" } EQ_Contact(in1 := "SN12_Step(ST10上)", in2 := 620)
      wire#w1
      I_Contact( "ST10上阻挡上到位" )
      Coil( "ST10上阻挡上指令自动" )
   END_RUNG
   RUNG wire#w1
      I_Contact( "AutoStep" )
      wire#w2
      Contact( "ST10上阻挡上到位" )
      Move(in := 699, out1 => "SN12_Step(ST10上)")
   END_RUNG
   RUNG wire#w1
      Contact( "AutoStep_P" )
   END_RUNG wire#w2
   // the same network as SCL:
   #_w1 := "Auto" AND ("SN12_Step(ST10上)" = 620);
   "ST10上阻挡上指令自动" := #_w1 AND NOT "ST10上阻挡上到位";
   IF #_w1 AND (NOT "AutoStep" OR "AutoStep_P") AND "ST10上阻挡上到位" THEN "SN12_Step(ST10上)" := 699; END_IF;
END_REGION

REGION Network 9: @返回
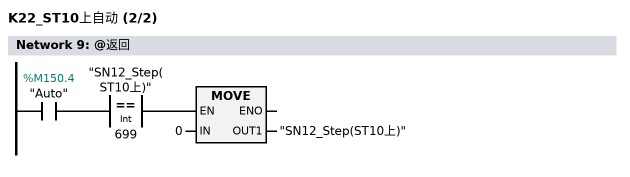
   RUNG wire#powerrail
      Contact( "Auto" )
      { S7_Templates := "SrcType := Int" } EQ_Contact(in1 := "SN12_Step(ST10上)", in2 := 699)
      Move(in := 0, out1 => "SN12_Step(ST10上)")
   END_RUNG
   // the same network as SCL:
   IF "Auto" AND ("SN12_Step(ST10上)" = 699) THEN "SN12_Step(ST10上)" := 0; END_IF;
END_REGION
END_FUNCTION_BLOCK

FUNCTION_BLOCK "K23_ST11上自动"   // FB23, LAD
{ S7_Optimized_Access := 'TRUE' }
VERSION : 0.1
// stored: AutoNumber false, IsIECCheckEnabled false, IsRetainMemResEnabled false, MemoryReserve 100, SetENOAutomatically false, UDAEnableTagReadback false
   VAR_TEMP   // added for the SCL form of the ladder/FBD networks
      _w1 : Bool;
   END_VAR
BEGIN

REGION Network 2: @搬出条件，SN13===ST11上工位
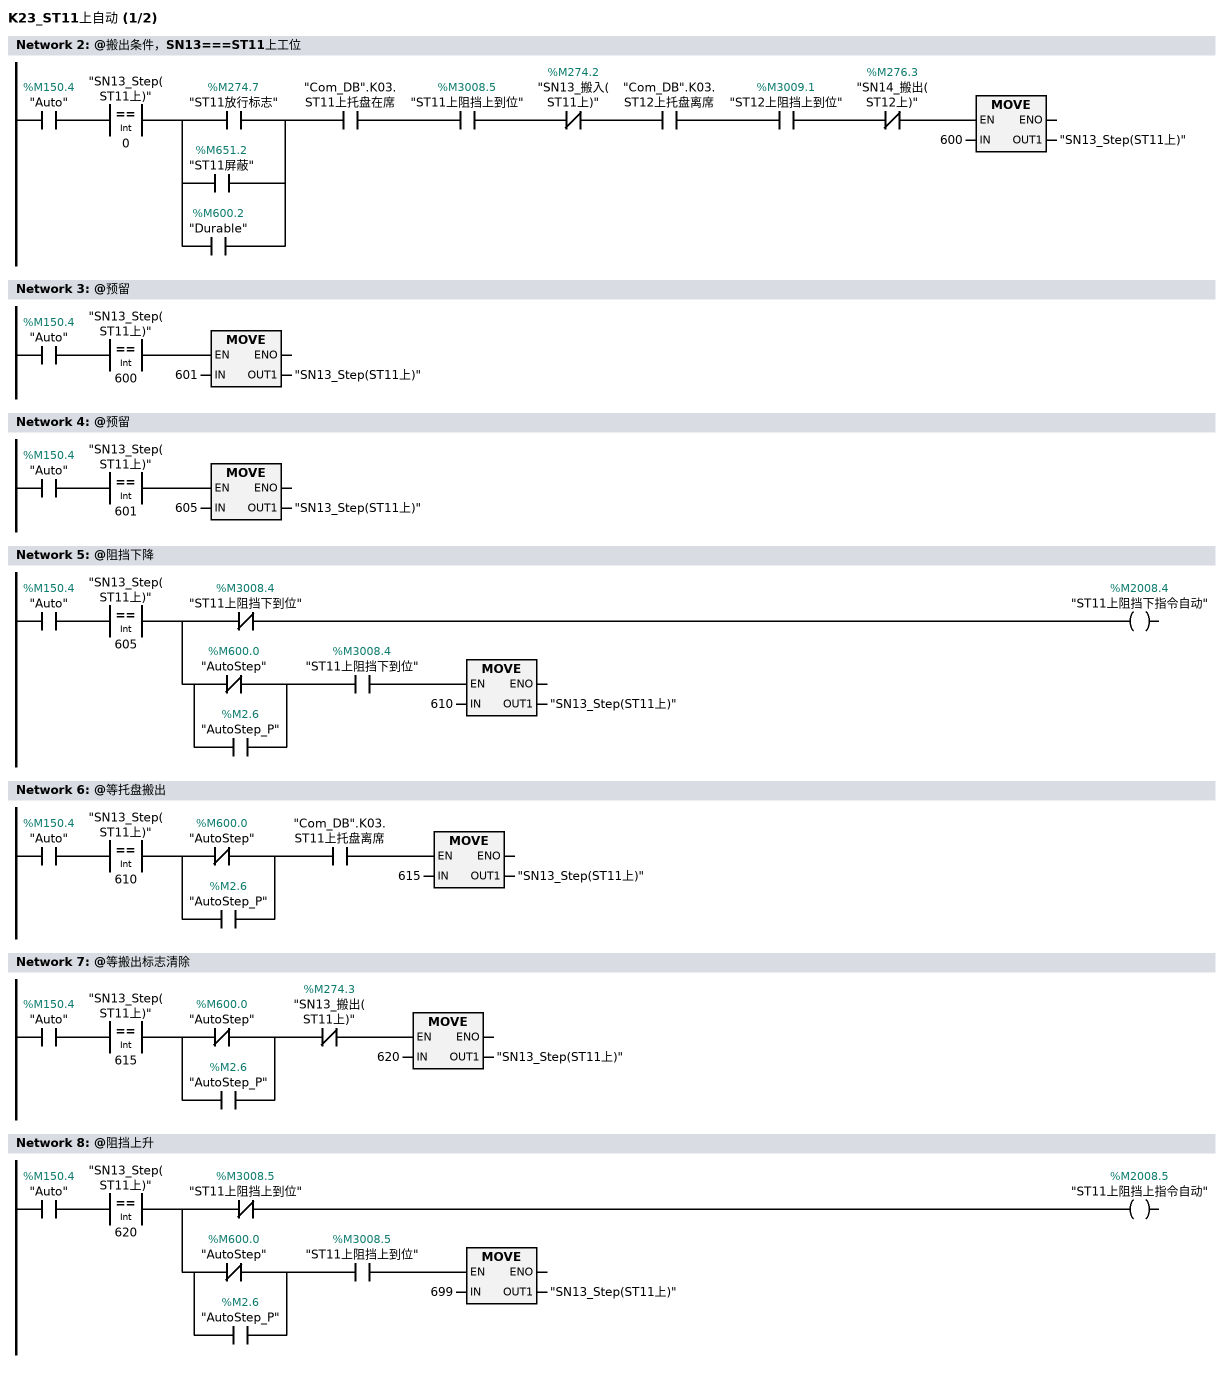
   RUNG wire#powerrail
      Contact( "Auto" )
      { S7_Templates := "SrcType := Int" } EQ_Contact(in1 := "SN13_Step(ST11上)", in2 := 0)
      wire#w1
      Contact( "ST11放行标志" )
      wire#w2
      Contact( "Com_DB".K03.ST11上托盘在席 )
      Contact( "ST11上阻挡上到位" )
      I_Contact( "SN13_搬入(ST11上)" )
      Contact( "Com_DB".K03.ST12上托盘离席 )
      Contact( "ST12上阻挡上到位" )
      I_Contact( "SN14_搬出(ST12上)" )
      Move(in := 600, out1 => "SN13_Step(ST11上)")
   END_RUNG
   RUNG wire#w1
      Contact( "ST11屏蔽" )
   END_RUNG wire#w2
   RUNG wire#w1
      Contact( "Durable" )
   END_RUNG wire#w2
   // the same network as SCL:
   IF "Auto" AND ("SN13_Step(ST11上)" = 0) AND ("ST11放行标志" OR "ST11屏蔽" OR "Durable") AND "Com_DB".K03.ST11上托盘在席 AND "ST11上阻挡上到位" AND NOT "SN13_搬入(ST11上)" AND "Com_DB".K03.ST12上托盘离席 AND "ST12上阻挡上到位" AND NOT "SN14_搬出(ST12上)" THEN
       "SN13_Step(ST11上)" := 600;
   END_IF;
END_REGION

REGION Network 3: @预留
   RUNG wire#powerrail
      Contact( "Auto" )
      { S7_Templates := "SrcType := Int" } EQ_Contact(in1 := "SN13_Step(ST11上)", in2 := 600)
      Move(in := 601, out1 => "SN13_Step(ST11上)")
   END_RUNG
   // the same network as SCL:
   IF "Auto" AND ("SN13_Step(ST11上)" = 600) THEN "SN13_Step(ST11上)" := 601; END_IF;
END_REGION

REGION Network 4: @预留
   RUNG wire#powerrail
      Contact( "Auto" )
      { S7_Templates := "SrcType := Int" } EQ_Contact(in1 := "SN13_Step(ST11上)", in2 := 601)
      Move(in := 605, out1 => "SN13_Step(ST11上)")
   END_RUNG
   // the same network as SCL:
   IF "Auto" AND ("SN13_Step(ST11上)" = 601) THEN "SN13_Step(ST11上)" := 605; END_IF;
END_REGION

REGION Network 5: @阻挡下降
   RUNG wire#powerrail
      Contact( "Auto" )
      { S7_Templates := "SrcType := Int" } EQ_Contact(in1 := "SN13_Step(ST11上)", in2 := 605)
      wire#w1
      I_Contact( "ST11上阻挡下到位" )
      Coil( "ST11上阻挡下指令自动" )
   END_RUNG
   RUNG wire#w1
      I_Contact( "AutoStep" )
      wire#w2
      Contact( "ST11上阻挡下到位" )
      Move(in := 610, out1 => "SN13_Step(ST11上)")
   END_RUNG
   RUNG wire#w1
      Contact( "AutoStep_P" )
   END_RUNG wire#w2
   // the same network as SCL:
   #_w1 := "Auto" AND ("SN13_Step(ST11上)" = 605);
   "ST11上阻挡下指令自动" := #_w1 AND NOT "ST11上阻挡下到位";
   IF #_w1 AND (NOT "AutoStep" OR "AutoStep_P") AND "ST11上阻挡下到位" THEN "SN13_Step(ST11上)" := 610; END_IF;
END_REGION

REGION Network 6: @等托盘搬出
   RUNG wire#powerrail
      Contact( "Auto" )
      { S7_Templates := "SrcType := Int" } EQ_Contact(in1 := "SN13_Step(ST11上)", in2 := 610)
      wire#w1
      I_Contact( "AutoStep" )
      wire#w2
      Contact( "Com_DB".K03.ST11上托盘离席 )
      Move(in := 615, out1 => "SN13_Step(ST11上)")
   END_RUNG
   RUNG wire#w1
      Contact( "AutoStep_P" )
   END_RUNG wire#w2
   // the same network as SCL:
   IF "Auto" AND ("SN13_Step(ST11上)" = 610) AND (NOT "AutoStep" OR "AutoStep_P") AND "Com_DB".K03.ST11上托盘离席 THEN
       "SN13_Step(ST11上)" := 615;
   END_IF;
END_REGION

REGION Network 7: @等搬出标志清除
   RUNG wire#powerrail
      Contact( "Auto" )
      { S7_Templates := "SrcType := Int" } EQ_Contact(in1 := "SN13_Step(ST11上)", in2 := 615)
      wire#w1
      I_Contact( "AutoStep" )
      wire#w2
      I_Contact( "SN13_搬出(ST11上)" )
      Move(in := 620, out1 => "SN13_Step(ST11上)")
   END_RUNG
   RUNG wire#w1
      Contact( "AutoStep_P" )
   END_RUNG wire#w2
   // the same network as SCL:
   IF "Auto" AND ("SN13_Step(ST11上)" = 615) AND (NOT "AutoStep" OR "AutoStep_P") AND NOT "SN13_搬出(ST11上)" THEN
       "SN13_Step(ST11上)" := 620;
   END_IF;
END_REGION

REGION Network 8: @阻挡上升
   RUNG wire#powerrail
      Contact( "Auto" )
      { S7_Templates := "SrcType := Int" } EQ_Contact(in1 := "SN13_Step(ST11上)", in2 := 620)
      wire#w1
      I_Contact( "ST11上阻挡上到位" )
      Coil( "ST11上阻挡上指令自动" )
   END_RUNG
   RUNG wire#w1
      I_Contact( "AutoStep" )
      wire#w2
      Contact( "ST11上阻挡上到位" )
      Move(in := 699, out1 => "SN13_Step(ST11上)")
   END_RUNG
   RUNG wire#w1
      Contact( "AutoStep_P" )
   END_RUNG wire#w2
   // the same network as SCL:
   #_w1 := "Auto" AND ("SN13_Step(ST11上)" = 620);
   "ST11上阻挡上指令自动" := #_w1 AND NOT "ST11上阻挡上到位";
   IF #_w1 AND (NOT "AutoStep" OR "AutoStep_P") AND "ST11上阻挡上到位" THEN "SN13_Step(ST11上)" := 699; END_IF;
END_REGION

REGION Network 9: @返回
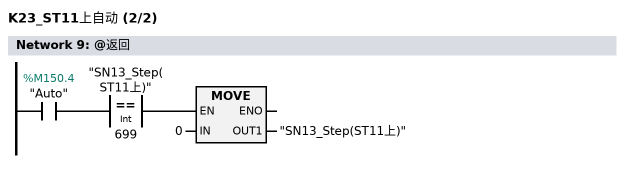
   RUNG wire#powerrail
      Contact( "Auto" )
      { S7_Templates := "SrcType := Int" } EQ_Contact(in1 := "SN13_Step(ST11上)", in2 := 699)
      Move(in := 0, out1 => "SN13_Step(ST11上)")
   END_RUNG
   // the same network as SCL:
   IF "Auto" AND ("SN13_Step(ST11上)" = 699) THEN "SN13_Step(ST11上)" := 0; END_IF;
END_REGION
END_FUNCTION_BLOCK

FUNCTION_BLOCK "K24_ST12上自动"   // FB24, LAD
{ S7_Optimized_Access := 'TRUE' }
VERSION : 0.1
// stored: AutoNumber false, IsIECCheckEnabled false, IsRetainMemResEnabled false, MemoryReserve 100, SetENOAutomatically false, UDAEnableTagReadback false
   VAR_TEMP   // added for the SCL form of the ladder/FBD networks
      _w1 : Bool;
   END_VAR
BEGIN

REGION Network 2: @搬出条件，SN14===ST12上工位
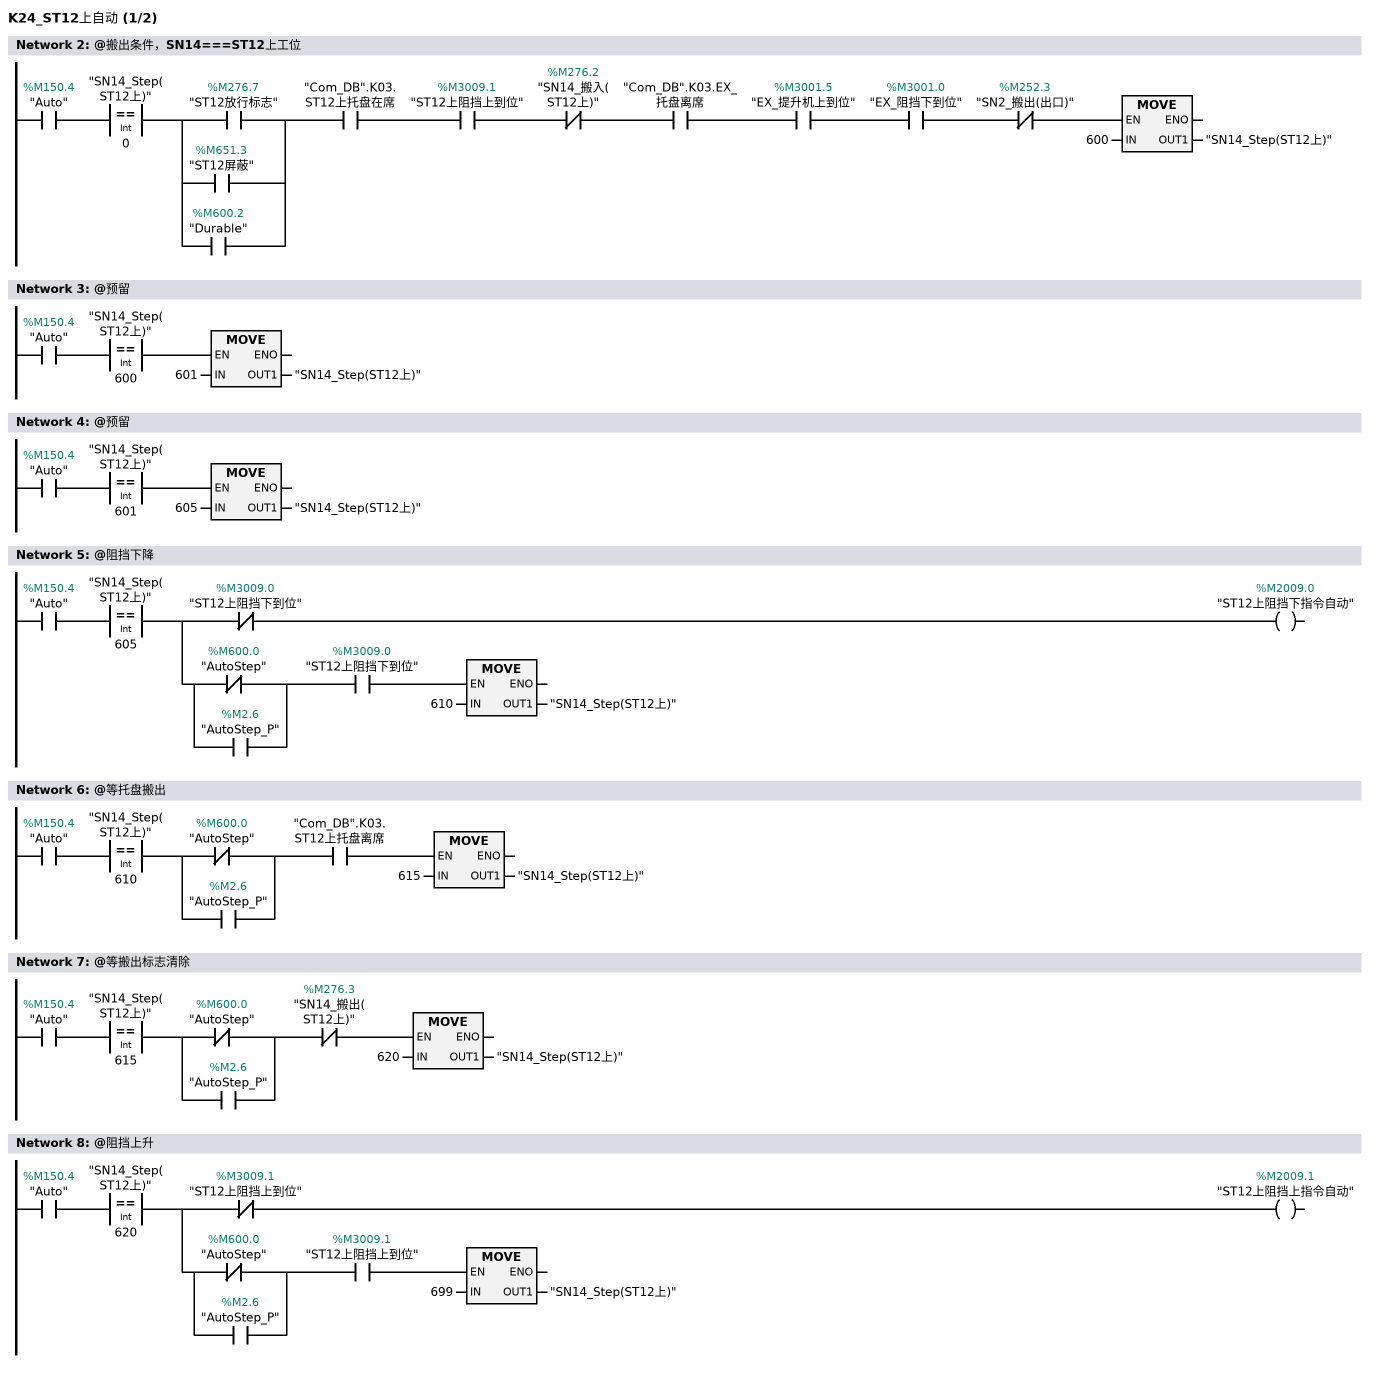
   RUNG wire#powerrail
      Contact( "Auto" )
      { S7_Templates := "SrcType := Int" } EQ_Contact(in1 := "SN14_Step(ST12上)", in2 := 0)
      wire#w1
      Contact( "ST12放行标志" )
      wire#w2
      Contact( "Com_DB".K03.ST12上托盘在席 )
      Contact( "ST12上阻挡上到位" )
      I_Contact( "SN14_搬入(ST12上)" )
      Contact( "Com_DB".K03.EX_托盘离席 )
      Contact( "EX_提升机上到位" )
      Contact( "EX_阻挡下到位" )
      I_Contact( "SN2_搬出(出口)" )
      Move(in := 600, out1 => "SN14_Step(ST12上)")
   END_RUNG
   RUNG wire#w1
      Contact( "ST12屏蔽" )
   END_RUNG wire#w2
   RUNG wire#w1
      Contact( "Durable" )
   END_RUNG wire#w2
   // the same network as SCL:
   IF "Auto" AND ("SN14_Step(ST12上)" = 0) AND ("ST12放行标志" OR "ST12屏蔽" OR "Durable") AND "Com_DB".K03.ST12上托盘在席 AND "ST12上阻挡上到位" AND NOT "SN14_搬入(ST12上)" AND "Com_DB".K03.EX_托盘离席 AND "EX_提升机上到位" AND "EX_阻挡下到位" AND NOT "SN2_搬出(出口)" THEN
       "SN14_Step(ST12上)" := 600;
   END_IF;
END_REGION

REGION Network 3: @预留
   RUNG wire#powerrail
      Contact( "Auto" )
      { S7_Templates := "SrcType := Int" } EQ_Contact(in1 := "SN14_Step(ST12上)", in2 := 600)
      Move(in := 601, out1 => "SN14_Step(ST12上)")
   END_RUNG
   // the same network as SCL:
   IF "Auto" AND ("SN14_Step(ST12上)" = 600) THEN "SN14_Step(ST12上)" := 601; END_IF;
END_REGION

REGION Network 4: @预留
   RUNG wire#powerrail
      Contact( "Auto" )
      { S7_Templates := "SrcType := Int" } EQ_Contact(in1 := "SN14_Step(ST12上)", in2 := 601)
      Move(in := 605, out1 => "SN14_Step(ST12上)")
   END_RUNG
   // the same network as SCL:
   IF "Auto" AND ("SN14_Step(ST12上)" = 601) THEN "SN14_Step(ST12上)" := 605; END_IF;
END_REGION

REGION Network 5: @阻挡下降
   RUNG wire#powerrail
      Contact( "Auto" )
      { S7_Templates := "SrcType := Int" } EQ_Contact(in1 := "SN14_Step(ST12上)", in2 := 605)
      wire#w1
      I_Contact( "ST12上阻挡下到位" )
      Coil( "ST12上阻挡下指令自动" )
   END_RUNG
   RUNG wire#w1
      I_Contact( "AutoStep" )
      wire#w2
      Contact( "ST12上阻挡下到位" )
      Move(in := 610, out1 => "SN14_Step(ST12上)")
   END_RUNG
   RUNG wire#w1
      Contact( "AutoStep_P" )
   END_RUNG wire#w2
   // the same network as SCL:
   #_w1 := "Auto" AND ("SN14_Step(ST12上)" = 605);
   "ST12上阻挡下指令自动" := #_w1 AND NOT "ST12上阻挡下到位";
   IF #_w1 AND (NOT "AutoStep" OR "AutoStep_P") AND "ST12上阻挡下到位" THEN "SN14_Step(ST12上)" := 610; END_IF;
END_REGION

REGION Network 6: @等托盘搬出
   RUNG wire#powerrail
      Contact( "Auto" )
      { S7_Templates := "SrcType := Int" } EQ_Contact(in1 := "SN14_Step(ST12上)", in2 := 610)
      wire#w1
      I_Contact( "AutoStep" )
      wire#w2
      Contact( "Com_DB".K03.ST12上托盘离席 )
      Move(in := 615, out1 => "SN14_Step(ST12上)")
   END_RUNG
   RUNG wire#w1
      Contact( "AutoStep_P" )
   END_RUNG wire#w2
   // the same network as SCL:
   IF "Auto" AND ("SN14_Step(ST12上)" = 610) AND (NOT "AutoStep" OR "AutoStep_P") AND "Com_DB".K03.ST12上托盘离席 THEN
       "SN14_Step(ST12上)" := 615;
   END_IF;
END_REGION

REGION Network 7: @等搬出标志清除
   RUNG wire#powerrail
      Contact( "Auto" )
      { S7_Templates := "SrcType := Int" } EQ_Contact(in1 := "SN14_Step(ST12上)", in2 := 615)
      wire#w1
      I_Contact( "AutoStep" )
      wire#w2
      I_Contact( "SN14_搬出(ST12上)" )
      Move(in := 620, out1 => "SN14_Step(ST12上)")
   END_RUNG
   RUNG wire#w1
      Contact( "AutoStep_P" )
   END_RUNG wire#w2
   // the same network as SCL:
   IF "Auto" AND ("SN14_Step(ST12上)" = 615) AND (NOT "AutoStep" OR "AutoStep_P") AND NOT "SN14_搬出(ST12上)" THEN
       "SN14_Step(ST12上)" := 620;
   END_IF;
END_REGION

REGION Network 8: @阻挡上升
   RUNG wire#powerrail
      Contact( "Auto" )
      { S7_Templates := "SrcType := Int" } EQ_Contact(in1 := "SN14_Step(ST12上)", in2 := 620)
      wire#w1
      I_Contact( "ST12上阻挡上到位" )
      Coil( "ST12上阻挡上指令自动" )
   END_RUNG
   RUNG wire#w1
      I_Contact( "AutoStep" )
      wire#w2
      Contact( "ST12上阻挡上到位" )
      Move(in := 699, out1 => "SN14_Step(ST12上)")
   END_RUNG
   RUNG wire#w1
      Contact( "AutoStep_P" )
   END_RUNG wire#w2
   // the same network as SCL:
   #_w1 := "Auto" AND ("SN14_Step(ST12上)" = 620);
   "ST12上阻挡上指令自动" := #_w1 AND NOT "ST12上阻挡上到位";
   IF #_w1 AND (NOT "AutoStep" OR "AutoStep_P") AND "ST12上阻挡上到位" THEN "SN14_Step(ST12上)" := 699; END_IF;
END_REGION

REGION Network 9: @返回
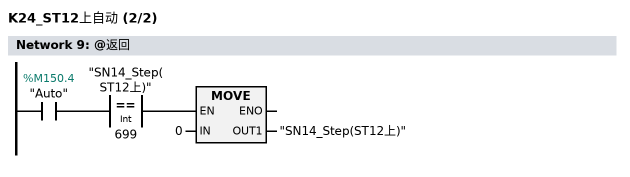
   RUNG wire#powerrail
      Contact( "Auto" )
      { S7_Templates := "SrcType := Int" } EQ_Contact(in1 := "SN14_Step(ST12上)", in2 := 699)
      Move(in := 0, out1 => "SN14_Step(ST12上)")
   END_RUNG
   // the same network as SCL:
   IF "Auto" AND ("SN14_Step(ST12上)" = 699) THEN "SN14_Step(ST12上)" := 0; END_IF;
END_REGION
END_FUNCTION_BLOCK

FUNCTION_BLOCK "K25_ST03下自动"   // FB25, LAD
{ S7_Optimized_Access := 'TRUE' }
VERSION : 0.1
// stored: AutoNumber false, IsIECCheckEnabled false, IsRetainMemResEnabled false, MemoryReserve 100, SetENOAutomatically false, UDAEnableTagReadback false
   VAR_TEMP   // added for the SCL form of the ladder/FBD networks
      _w1 : Bool;
   END_VAR
BEGIN

REGION Network 2: @搬出条件，SN15===ST03下工位
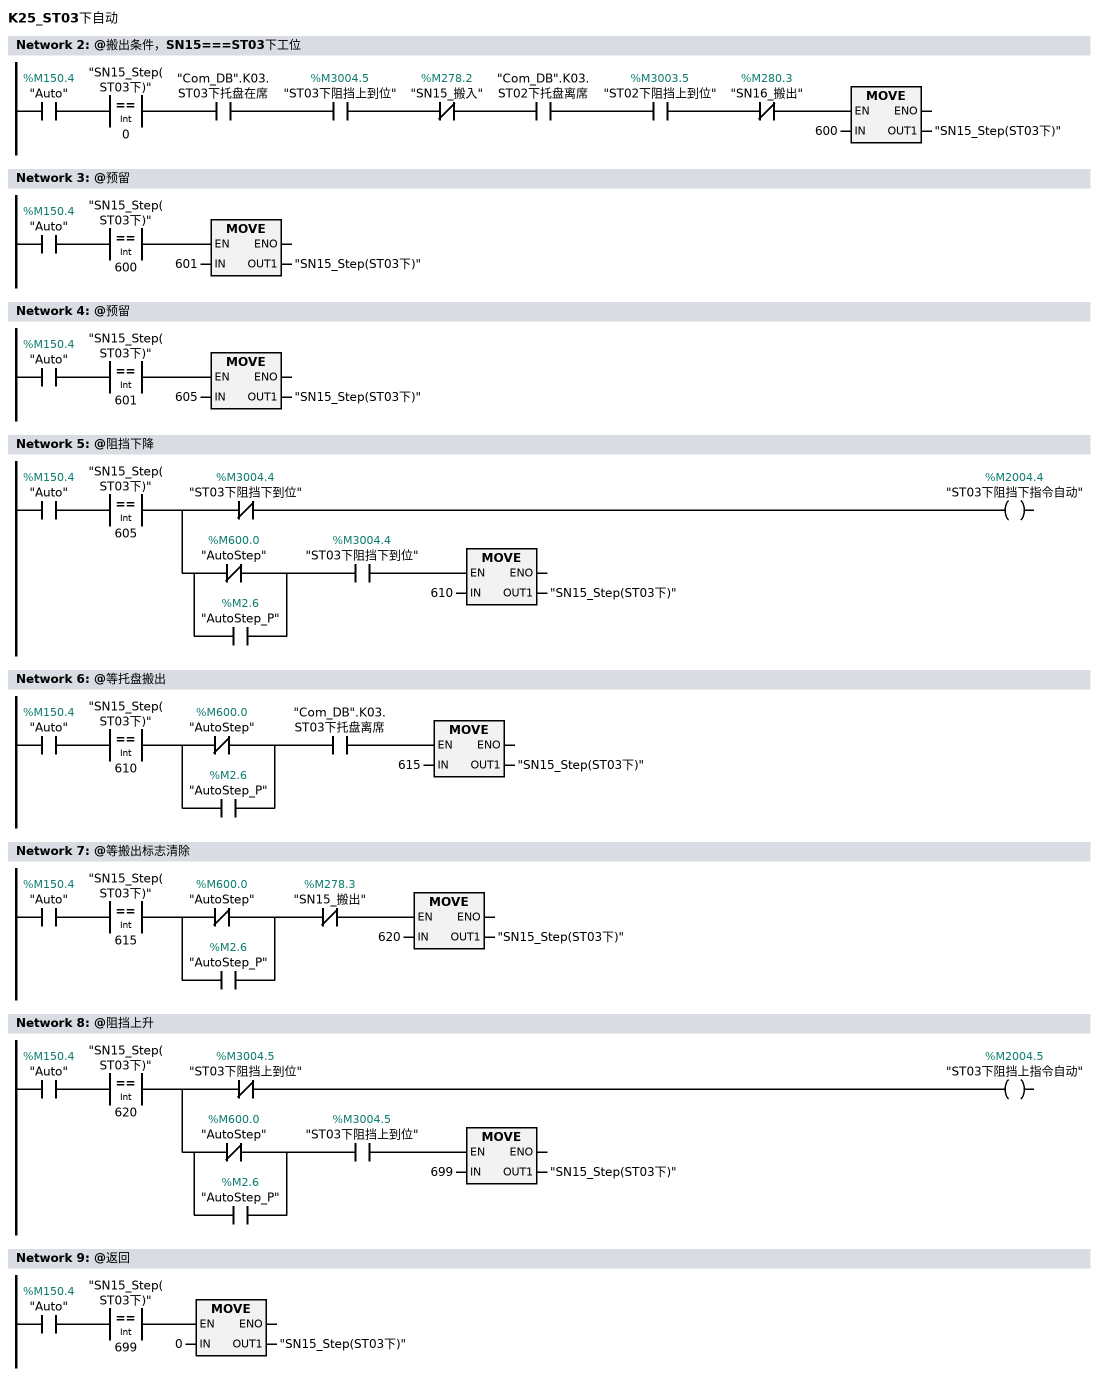
   RUNG wire#powerrail
      Contact( "Auto" )
      { S7_Templates := "SrcType := Int" } EQ_Contact(in1 := "SN15_Step(ST03下)", in2 := 0)
      Contact( "Com_DB".K03.ST03下托盘在席 )
      Contact( "ST03下阻挡上到位" )
      I_Contact( "SN15_搬入" )
      Contact( "Com_DB".K03.ST02下托盘离席 )
      Contact( "ST02下阻挡上到位" )
      I_Contact( "SN16_搬出" )
      Move(in := 600, out1 => "SN15_Step(ST03下)")
   END_RUNG
   // the same network as SCL:
   IF "Auto" AND ("SN15_Step(ST03下)" = 0) AND "Com_DB".K03.ST03下托盘在席 AND "ST03下阻挡上到位" AND NOT "SN15_搬入" AND "Com_DB".K03.ST02下托盘离席 AND "ST02下阻挡上到位" AND NOT "SN16_搬出" THEN
       "SN15_Step(ST03下)" := 600;
   END_IF;
END_REGION

REGION Network 3: @预留
   RUNG wire#powerrail
      Contact( "Auto" )
      { S7_Templates := "SrcType := Int" } EQ_Contact(in1 := "SN15_Step(ST03下)", in2 := 600)
      Move(in := 601, out1 => "SN15_Step(ST03下)")
   END_RUNG
   // the same network as SCL:
   IF "Auto" AND ("SN15_Step(ST03下)" = 600) THEN "SN15_Step(ST03下)" := 601; END_IF;
END_REGION

REGION Network 4: @预留
   RUNG wire#powerrail
      Contact( "Auto" )
      { S7_Templates := "SrcType := Int" } EQ_Contact(in1 := "SN15_Step(ST03下)", in2 := 601)
      Move(in := 605, out1 => "SN15_Step(ST03下)")
   END_RUNG
   // the same network as SCL:
   IF "Auto" AND ("SN15_Step(ST03下)" = 601) THEN "SN15_Step(ST03下)" := 605; END_IF;
END_REGION

REGION Network 5: @阻挡下降
   RUNG wire#powerrail
      Contact( "Auto" )
      { S7_Templates := "SrcType := Int" } EQ_Contact(in1 := "SN15_Step(ST03下)", in2 := 605)
      wire#w1
      I_Contact( "ST03下阻挡下到位" )
      Coil( "ST03下阻挡下指令自动" )
   END_RUNG
   RUNG wire#w1
      I_Contact( "AutoStep" )
      wire#w2
      Contact( "ST03下阻挡下到位" )
      Move(in := 610, out1 => "SN15_Step(ST03下)")
   END_RUNG
   RUNG wire#w1
      Contact( "AutoStep_P" )
   END_RUNG wire#w2
   // the same network as SCL:
   #_w1 := "Auto" AND ("SN15_Step(ST03下)" = 605);
   "ST03下阻挡下指令自动" := #_w1 AND NOT "ST03下阻挡下到位";
   IF #_w1 AND (NOT "AutoStep" OR "AutoStep_P") AND "ST03下阻挡下到位" THEN "SN15_Step(ST03下)" := 610; END_IF;
END_REGION

REGION Network 6: @等托盘搬出
   RUNG wire#powerrail
      Contact( "Auto" )
      { S7_Templates := "SrcType := Int" } EQ_Contact(in1 := "SN15_Step(ST03下)", in2 := 610)
      wire#w1
      I_Contact( "AutoStep" )
      wire#w2
      Contact( "Com_DB".K03.ST03下托盘离席 )
      Move(in := 615, out1 => "SN15_Step(ST03下)")
   END_RUNG
   RUNG wire#w1
      Contact( "AutoStep_P" )
   END_RUNG wire#w2
   // the same network as SCL:
   IF "Auto" AND ("SN15_Step(ST03下)" = 610) AND (NOT "AutoStep" OR "AutoStep_P") AND "Com_DB".K03.ST03下托盘离席 THEN
       "SN15_Step(ST03下)" := 615;
   END_IF;
END_REGION

REGION Network 7: @等搬出标志清除
   RUNG wire#powerrail
      Contact( "Auto" )
      { S7_Templates := "SrcType := Int" } EQ_Contact(in1 := "SN15_Step(ST03下)", in2 := 615)
      wire#w1
      I_Contact( "AutoStep" )
      wire#w2
      I_Contact( "SN15_搬出" )
      Move(in := 620, out1 => "SN15_Step(ST03下)")
   END_RUNG
   RUNG wire#w1
      Contact( "AutoStep_P" )
   END_RUNG wire#w2
   // the same network as SCL:
   IF "Auto" AND ("SN15_Step(ST03下)" = 615) AND (NOT "AutoStep" OR "AutoStep_P") AND NOT "SN15_搬出" THEN
       "SN15_Step(ST03下)" := 620;
   END_IF;
END_REGION

REGION Network 8: @阻挡上升
   RUNG wire#powerrail
      Contact( "Auto" )
      { S7_Templates := "SrcType := Int" } EQ_Contact(in1 := "SN15_Step(ST03下)", in2 := 620)
      wire#w1
      I_Contact( "ST03下阻挡上到位" )
      Coil( "ST03下阻挡上指令自动" )
   END_RUNG
   RUNG wire#w1
      I_Contact( "AutoStep" )
      wire#w2
      Contact( "ST03下阻挡上到位" )
      Move(in := 699, out1 => "SN15_Step(ST03下)")
   END_RUNG
   RUNG wire#w1
      Contact( "AutoStep_P" )
   END_RUNG wire#w2
   // the same network as SCL:
   #_w1 := "Auto" AND ("SN15_Step(ST03下)" = 620);
   "ST03下阻挡上指令自动" := #_w1 AND NOT "ST03下阻挡上到位";
   IF #_w1 AND (NOT "AutoStep" OR "AutoStep_P") AND "ST03下阻挡上到位" THEN "SN15_Step(ST03下)" := 699; END_IF;
END_REGION

REGION Network 9: @返回
   RUNG wire#powerrail
      Contact( "Auto" )
      { S7_Templates := "SrcType := Int" } EQ_Contact(in1 := "SN15_Step(ST03下)", in2 := 699)
      Move(in := 0, out1 => "SN15_Step(ST03下)")
   END_RUNG
   // the same network as SCL:
   IF "Auto" AND ("SN15_Step(ST03下)" = 699) THEN "SN15_Step(ST03下)" := 0; END_IF;
END_REGION
END_FUNCTION_BLOCK

FUNCTION_BLOCK "K26_ST02下自动"   // FB26, LAD
{ S7_Optimized_Access := 'TRUE' }
VERSION : 0.1
// stored: AutoNumber false, IsIECCheckEnabled false, IsRetainMemResEnabled false, MemoryReserve 100, SetENOAutomatically false, UDAEnableTagReadback false
   VAR_TEMP   // added for the SCL form of the ladder/FBD networks
      _w1 : Bool;
   END_VAR
BEGIN

REGION Network 2: @搬出条件，SN16===ST02下工位
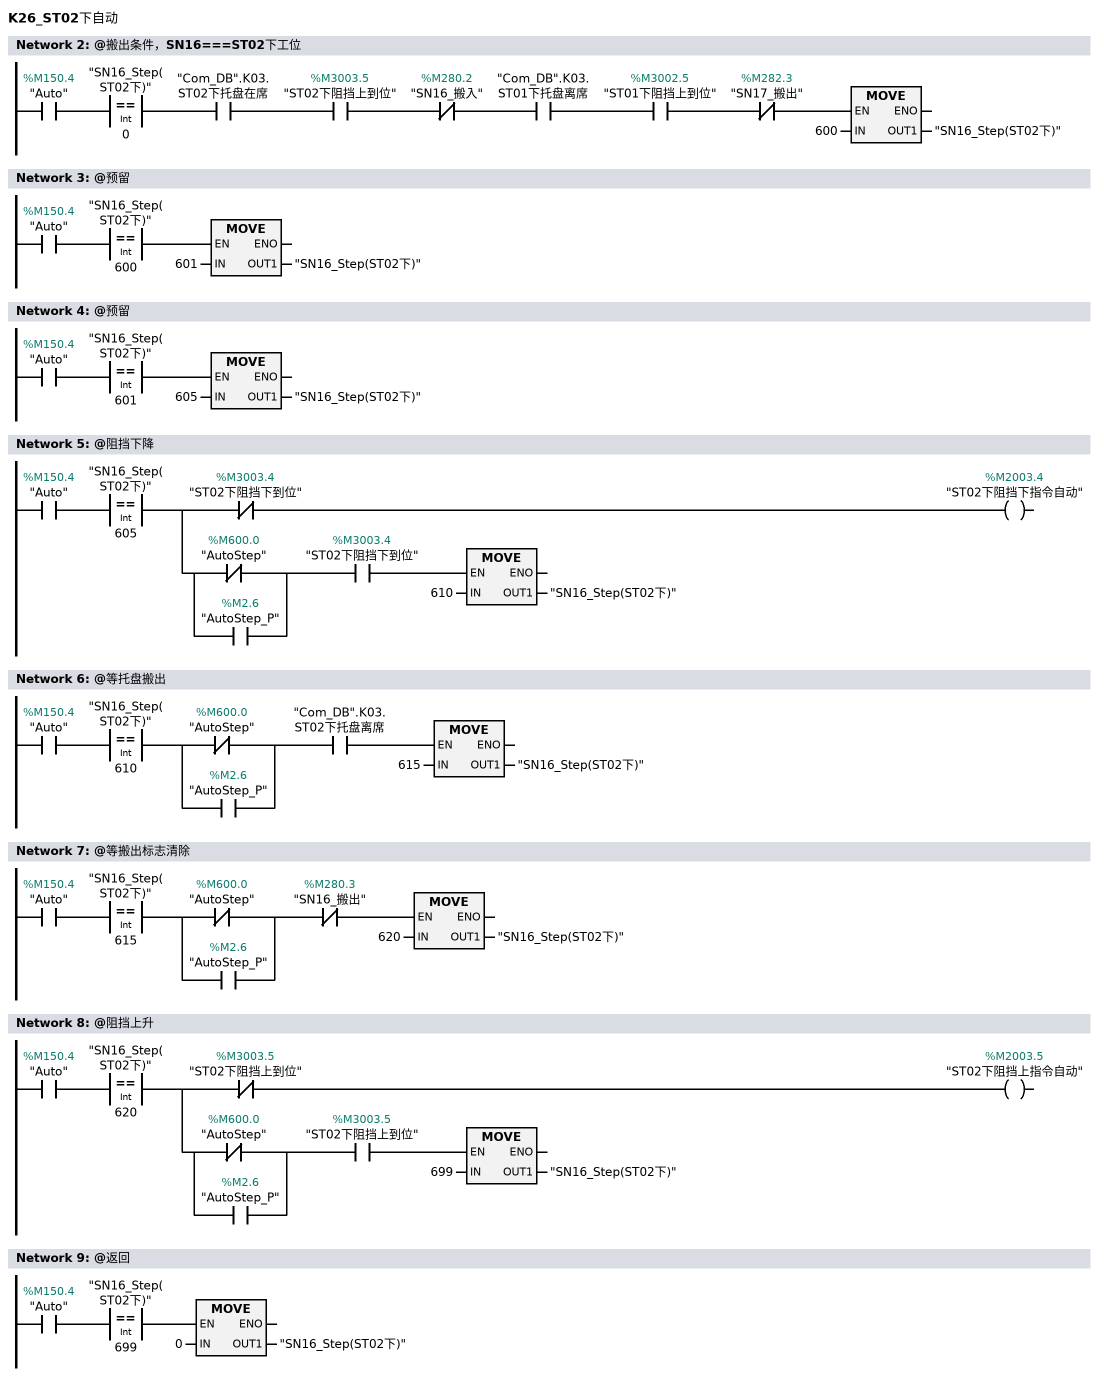
   RUNG wire#powerrail
      Contact( "Auto" )
      { S7_Templates := "SrcType := Int" } EQ_Contact(in1 := "SN16_Step(ST02下)", in2 := 0)
      Contact( "Com_DB".K03.ST02下托盘在席 )
      Contact( "ST02下阻挡上到位" )
      I_Contact( "SN16_搬入" )
      Contact( "Com_DB".K03.ST01下托盘离席 )
      Contact( "ST01下阻挡上到位" )
      I_Contact( "SN17_搬出" )
      Move(in := 600, out1 => "SN16_Step(ST02下)")
   END_RUNG
   // the same network as SCL:
   IF "Auto" AND ("SN16_Step(ST02下)" = 0) AND "Com_DB".K03.ST02下托盘在席 AND "ST02下阻挡上到位" AND NOT "SN16_搬入" AND "Com_DB".K03.ST01下托盘离席 AND "ST01下阻挡上到位" AND NOT "SN17_搬出" THEN
       "SN16_Step(ST02下)" := 600;
   END_IF;
END_REGION

REGION Network 3: @预留
   RUNG wire#powerrail
      Contact( "Auto" )
      { S7_Templates := "SrcType := Int" } EQ_Contact(in1 := "SN16_Step(ST02下)", in2 := 600)
      Move(in := 601, out1 => "SN16_Step(ST02下)")
   END_RUNG
   // the same network as SCL:
   IF "Auto" AND ("SN16_Step(ST02下)" = 600) THEN "SN16_Step(ST02下)" := 601; END_IF;
END_REGION

REGION Network 4: @预留
   RUNG wire#powerrail
      Contact( "Auto" )
      { S7_Templates := "SrcType := Int" } EQ_Contact(in1 := "SN16_Step(ST02下)", in2 := 601)
      Move(in := 605, out1 => "SN16_Step(ST02下)")
   END_RUNG
   // the same network as SCL:
   IF "Auto" AND ("SN16_Step(ST02下)" = 601) THEN "SN16_Step(ST02下)" := 605; END_IF;
END_REGION

REGION Network 5: @阻挡下降
   RUNG wire#powerrail
      Contact( "Auto" )
      { S7_Templates := "SrcType := Int" } EQ_Contact(in1 := "SN16_Step(ST02下)", in2 := 605)
      wire#w1
      I_Contact( "ST02下阻挡下到位" )
      Coil( "ST02下阻挡下指令自动" )
   END_RUNG
   RUNG wire#w1
      I_Contact( "AutoStep" )
      wire#w2
      Contact( "ST02下阻挡下到位" )
      Move(in := 610, out1 => "SN16_Step(ST02下)")
   END_RUNG
   RUNG wire#w1
      Contact( "AutoStep_P" )
   END_RUNG wire#w2
   // the same network as SCL:
   #_w1 := "Auto" AND ("SN16_Step(ST02下)" = 605);
   "ST02下阻挡下指令自动" := #_w1 AND NOT "ST02下阻挡下到位";
   IF #_w1 AND (NOT "AutoStep" OR "AutoStep_P") AND "ST02下阻挡下到位" THEN "SN16_Step(ST02下)" := 610; END_IF;
END_REGION

REGION Network 6: @等托盘搬出
   RUNG wire#powerrail
      Contact( "Auto" )
      { S7_Templates := "SrcType := Int" } EQ_Contact(in1 := "SN16_Step(ST02下)", in2 := 610)
      wire#w1
      I_Contact( "AutoStep" )
      wire#w2
      Contact( "Com_DB".K03.ST02下托盘离席 )
      Move(in := 615, out1 => "SN16_Step(ST02下)")
   END_RUNG
   RUNG wire#w1
      Contact( "AutoStep_P" )
   END_RUNG wire#w2
   // the same network as SCL:
   IF "Auto" AND ("SN16_Step(ST02下)" = 610) AND (NOT "AutoStep" OR "AutoStep_P") AND "Com_DB".K03.ST02下托盘离席 THEN
       "SN16_Step(ST02下)" := 615;
   END_IF;
END_REGION

REGION Network 7: @等搬出标志清除
   RUNG wire#powerrail
      Contact( "Auto" )
      { S7_Templates := "SrcType := Int" } EQ_Contact(in1 := "SN16_Step(ST02下)", in2 := 615)
      wire#w1
      I_Contact( "AutoStep" )
      wire#w2
      I_Contact( "SN16_搬出" )
      Move(in := 620, out1 => "SN16_Step(ST02下)")
   END_RUNG
   RUNG wire#w1
      Contact( "AutoStep_P" )
   END_RUNG wire#w2
   // the same network as SCL:
   IF "Auto" AND ("SN16_Step(ST02下)" = 615) AND (NOT "AutoStep" OR "AutoStep_P") AND NOT "SN16_搬出" THEN
       "SN16_Step(ST02下)" := 620;
   END_IF;
END_REGION

REGION Network 8: @阻挡上升
   RUNG wire#powerrail
      Contact( "Auto" )
      { S7_Templates := "SrcType := Int" } EQ_Contact(in1 := "SN16_Step(ST02下)", in2 := 620)
      wire#w1
      I_Contact( "ST02下阻挡上到位" )
      Coil( "ST02下阻挡上指令自动" )
   END_RUNG
   RUNG wire#w1
      I_Contact( "AutoStep" )
      wire#w2
      Contact( "ST02下阻挡上到位" )
      Move(in := 699, out1 => "SN16_Step(ST02下)")
   END_RUNG
   RUNG wire#w1
      Contact( "AutoStep_P" )
   END_RUNG wire#w2
   // the same network as SCL:
   #_w1 := "Auto" AND ("SN16_Step(ST02下)" = 620);
   "ST02下阻挡上指令自动" := #_w1 AND NOT "ST02下阻挡上到位";
   IF #_w1 AND (NOT "AutoStep" OR "AutoStep_P") AND "ST02下阻挡上到位" THEN "SN16_Step(ST02下)" := 699; END_IF;
END_REGION

REGION Network 9: @返回
   RUNG wire#powerrail
      Contact( "Auto" )
      { S7_Templates := "SrcType := Int" } EQ_Contact(in1 := "SN16_Step(ST02下)", in2 := 699)
      Move(in := 0, out1 => "SN16_Step(ST02下)")
   END_RUNG
   // the same network as SCL:
   IF "Auto" AND ("SN16_Step(ST02下)" = 699) THEN "SN16_Step(ST02下)" := 0; END_IF;
END_REGION
END_FUNCTION_BLOCK

FUNCTION_BLOCK "K27_ST01下自动"   // FB27, LAD
{ S7_Optimized_Access := 'TRUE' }
VERSION : 0.1
// stored: AutoNumber false, IsIECCheckEnabled false, IsRetainMemResEnabled false, MemoryReserve 100, SetENOAutomatically false, UDAEnableTagReadback false
   VAR_TEMP   // added for the SCL form of the ladder/FBD networks
      _w1 : Bool;
   END_VAR
BEGIN

REGION Network 2: @搬出条件，SN17===ST01下工位
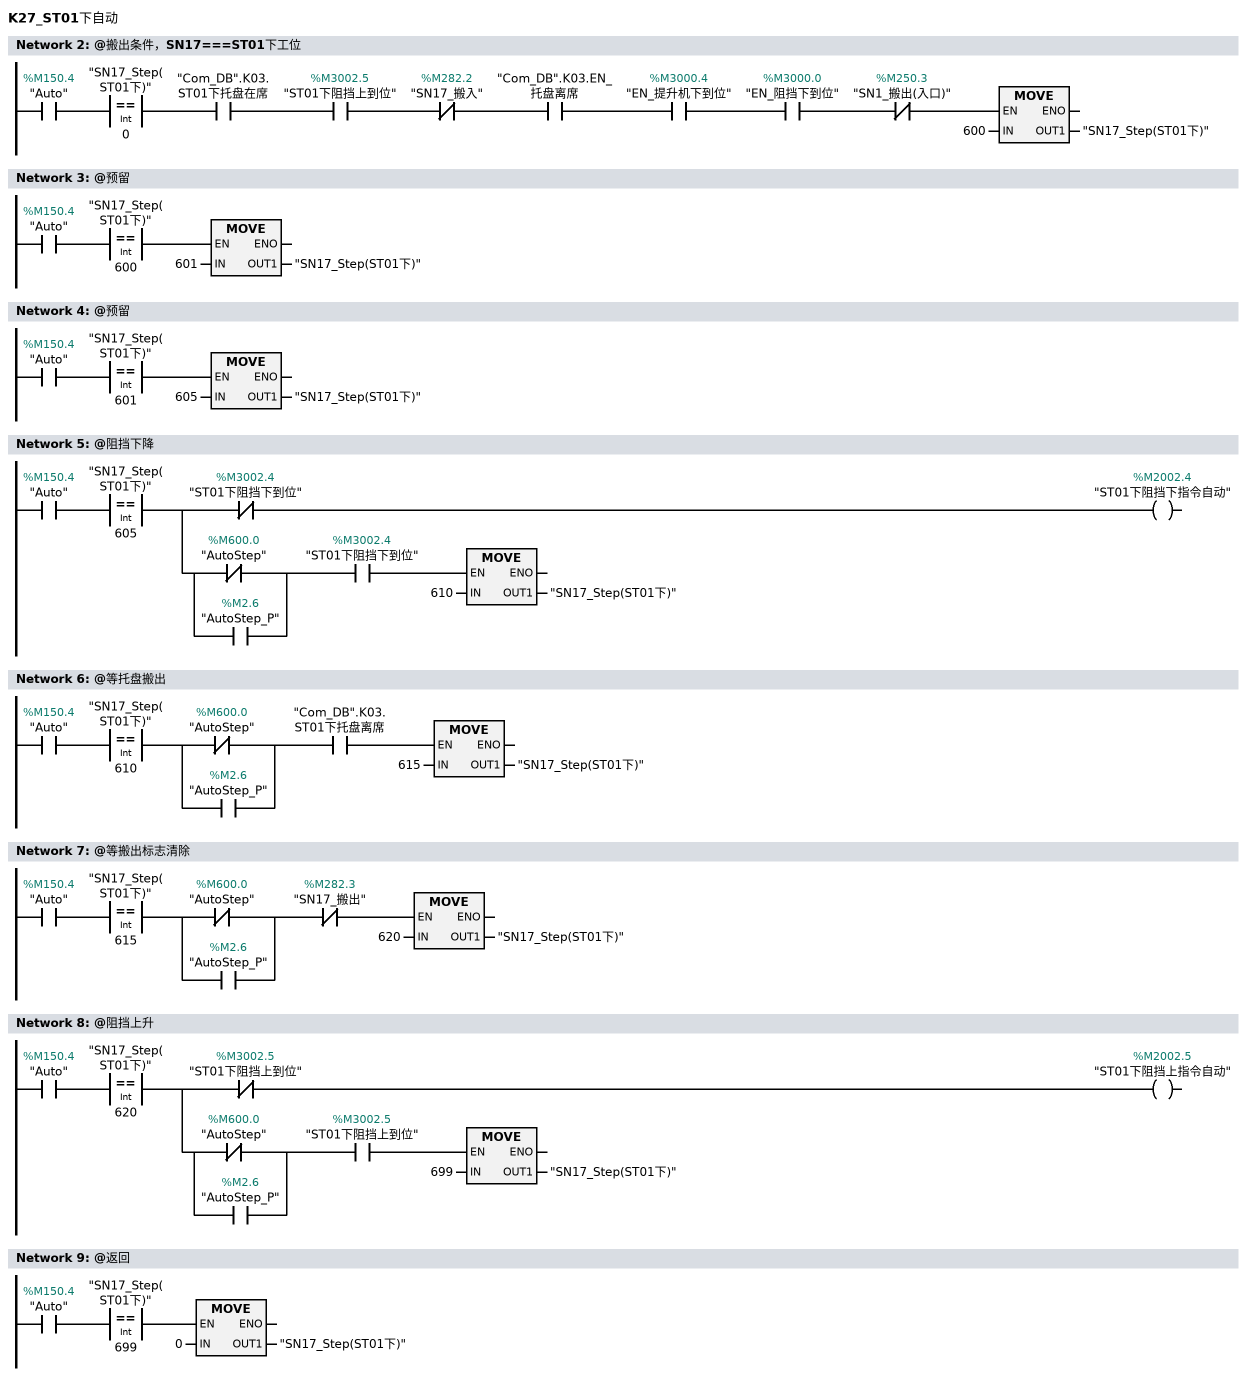
   RUNG wire#powerrail
      Contact( "Auto" )
      { S7_Templates := "SrcType := Int" } EQ_Contact(in1 := "SN17_Step(ST01下)", in2 := 0)
      Contact( "Com_DB".K03.ST01下托盘在席 )
      Contact( "ST01下阻挡上到位" )
      I_Contact( "SN17_搬入" )
      Contact( "Com_DB".K03.EN_托盘离席 )
      Contact( "EN_提升机下到位" )
      Contact( "EN_阻挡下到位" )
      I_Contact( "SN1_搬出(入口)" )
      Move(in := 600, out1 => "SN17_Step(ST01下)")
   END_RUNG
   // the same network as SCL:
   IF "Auto" AND ("SN17_Step(ST01下)" = 0) AND "Com_DB".K03.ST01下托盘在席 AND "ST01下阻挡上到位" AND NOT "SN17_搬入" AND "Com_DB".K03.EN_托盘离席 AND "EN_提升机下到位" AND "EN_阻挡下到位" AND NOT "SN1_搬出(入口)" THEN
       "SN17_Step(ST01下)" := 600;
   END_IF;
END_REGION

REGION Network 3: @预留
   RUNG wire#powerrail
      Contact( "Auto" )
      { S7_Templates := "SrcType := Int" } EQ_Contact(in1 := "SN17_Step(ST01下)", in2 := 600)
      Move(in := 601, out1 => "SN17_Step(ST01下)")
   END_RUNG
   // the same network as SCL:
   IF "Auto" AND ("SN17_Step(ST01下)" = 600) THEN "SN17_Step(ST01下)" := 601; END_IF;
END_REGION

REGION Network 4: @预留
   RUNG wire#powerrail
      Contact( "Auto" )
      { S7_Templates := "SrcType := Int" } EQ_Contact(in1 := "SN17_Step(ST01下)", in2 := 601)
      Move(in := 605, out1 => "SN17_Step(ST01下)")
   END_RUNG
   // the same network as SCL:
   IF "Auto" AND ("SN17_Step(ST01下)" = 601) THEN "SN17_Step(ST01下)" := 605; END_IF;
END_REGION

REGION Network 5: @阻挡下降
   RUNG wire#powerrail
      Contact( "Auto" )
      { S7_Templates := "SrcType := Int" } EQ_Contact(in1 := "SN17_Step(ST01下)", in2 := 605)
      wire#w1
      I_Contact( "ST01下阻挡下到位" )
      Coil( "ST01下阻挡下指令自动" )
   END_RUNG
   RUNG wire#w1
      I_Contact( "AutoStep" )
      wire#w2
      Contact( "ST01下阻挡下到位" )
      Move(in := 610, out1 => "SN17_Step(ST01下)")
   END_RUNG
   RUNG wire#w1
      Contact( "AutoStep_P" )
   END_RUNG wire#w2
   // the same network as SCL:
   #_w1 := "Auto" AND ("SN17_Step(ST01下)" = 605);
   "ST01下阻挡下指令自动" := #_w1 AND NOT "ST01下阻挡下到位";
   IF #_w1 AND (NOT "AutoStep" OR "AutoStep_P") AND "ST01下阻挡下到位" THEN "SN17_Step(ST01下)" := 610; END_IF;
END_REGION

REGION Network 6: @等托盘搬出
   RUNG wire#powerrail
      Contact( "Auto" )
      { S7_Templates := "SrcType := Int" } EQ_Contact(in1 := "SN17_Step(ST01下)", in2 := 610)
      wire#w1
      I_Contact( "AutoStep" )
      wire#w2
      Contact( "Com_DB".K03.ST01下托盘离席 )
      Move(in := 615, out1 => "SN17_Step(ST01下)")
   END_RUNG
   RUNG wire#w1
      Contact( "AutoStep_P" )
   END_RUNG wire#w2
   // the same network as SCL:
   IF "Auto" AND ("SN17_Step(ST01下)" = 610) AND (NOT "AutoStep" OR "AutoStep_P") AND "Com_DB".K03.ST01下托盘离席 THEN
       "SN17_Step(ST01下)" := 615;
   END_IF;
END_REGION

REGION Network 7: @等搬出标志清除
   RUNG wire#powerrail
      Contact( "Auto" )
      { S7_Templates := "SrcType := Int" } EQ_Contact(in1 := "SN17_Step(ST01下)", in2 := 615)
      wire#w1
      I_Contact( "AutoStep" )
      wire#w2
      I_Contact( "SN17_搬出" )
      Move(in := 620, out1 => "SN17_Step(ST01下)")
   END_RUNG
   RUNG wire#w1
      Contact( "AutoStep_P" )
   END_RUNG wire#w2
   // the same network as SCL:
   IF "Auto" AND ("SN17_Step(ST01下)" = 615) AND (NOT "AutoStep" OR "AutoStep_P") AND NOT "SN17_搬出" THEN
       "SN17_Step(ST01下)" := 620;
   END_IF;
END_REGION

REGION Network 8: @阻挡上升
   RUNG wire#powerrail
      Contact( "Auto" )
      { S7_Templates := "SrcType := Int" } EQ_Contact(in1 := "SN17_Step(ST01下)", in2 := 620)
      wire#w1
      I_Contact( "ST01下阻挡上到位" )
      Coil( "ST01下阻挡上指令自动" )
   END_RUNG
   RUNG wire#w1
      I_Contact( "AutoStep" )
      wire#w2
      Contact( "ST01下阻挡上到位" )
      Move(in := 699, out1 => "SN17_Step(ST01下)")
   END_RUNG
   RUNG wire#w1
      Contact( "AutoStep_P" )
   END_RUNG wire#w2
   // the same network as SCL:
   #_w1 := "Auto" AND ("SN17_Step(ST01下)" = 620);
   "ST01下阻挡上指令自动" := #_w1 AND NOT "ST01下阻挡上到位";
   IF #_w1 AND (NOT "AutoStep" OR "AutoStep_P") AND "ST01下阻挡上到位" THEN "SN17_Step(ST01下)" := 699; END_IF;
END_REGION

REGION Network 9: @返回
   RUNG wire#powerrail
      Contact( "Auto" )
      { S7_Templates := "SrcType := Int" } EQ_Contact(in1 := "SN17_Step(ST01下)", in2 := 699)
      Move(in := 0, out1 => "SN17_Step(ST01下)")
   END_RUNG
   // the same network as SCL:
   IF "Auto" AND ("SN17_Step(ST01下)" = 699) THEN "SN17_Step(ST01下)" := 0; END_IF;
END_REGION
END_FUNCTION_BLOCK

FUNCTION_BLOCK "K40_互锁"   // FB40, LAD
{ S7_Optimized_Access := 'TRUE' }
VERSION : 0.1
// stored: AutoNumber false, IsIECCheckEnabled false, IsRetainMemResEnabled false, MemoryReserve 100, SetENOAutomatically false, UDAEnableTagReadback false
BEGIN
END_FUNCTION_BLOCK

DATA_BLOCK "K08_指示灯_DB"   // DB8
VERSION : 0.1
// stored: AutoNumber false, DBAccessibleFromOPCUA true, InstanceOfName K08_指示灯, InstanceOfType FB
"K08_指示灯"
BEGIN
END_DATA_BLOCK

DATA_BLOCK "K02_初始化_DB"   // DB2
VERSION : 0.1
// stored: AutoNumber true, DBAccessibleFromOPCUA true, InstanceOfName K02_初始化, InstanceOfType FB
"K02_初始化"
BEGIN
END_DATA_BLOCK

DATA_BLOCK "K03_状态_DB"   // DB3
VERSION : 0.1
// stored: AutoNumber true, DBAccessibleFromOPCUA true, InstanceOfName K03_状态, InstanceOfType FB
"K03_状态"
BEGIN
END_DATA_BLOCK

DATA_BLOCK "K04_报警_DB"   // DB4
VERSION : 0.1
// stored: AutoNumber true, DBAccessibleFromOPCUA true, InstanceOfName K04_报警, InstanceOfType FB
"K04_报警"
BEGIN
END_DATA_BLOCK

DATA_BLOCK "K05_模式_DB"   // DB5
VERSION : 0.1
// stored: AutoNumber true, DBAccessibleFromOPCUA true, InstanceOfName K05_模式, InstanceOfType FB
"K05_模式"
BEGIN
END_DATA_BLOCK

DATA_BLOCK "K06_动作_DB"   // DB6
VERSION : 0.1
// stored: AutoNumber true, DBAccessibleFromOPCUA true, InstanceOfName K06_动作, InstanceOfType FB
"K06_动作"
BEGIN
END_DATA_BLOCK

DATA_BLOCK "K07_轴组_DB"   // DB7
VERSION : 0.1
// stored: AutoNumber true, DBAccessibleFromOPCUA true, InstanceOfName K07_轴组, InstanceOfType FB
"K07_轴组"
BEGIN
END_DATA_BLOCK

DATA_BLOCK "K10_自动_DB"   // DB10
VERSION : 0.1
// stored: AutoNumber false, DBAccessibleFromOPCUA true, InstanceOfName K10_自动, InstanceOfType FB
"K10_自动"
BEGIN
END_DATA_BLOCK

DATA_BLOCK "K11_入口自动_DB"   // DB11
VERSION : 0.1
// stored: AutoNumber false, DBAccessibleFromOPCUA true, InstanceOfName K11_入口自动, InstanceOfType FB
"K11_入口自动"
BEGIN
END_DATA_BLOCK

DATA_BLOCK "K12_出口自动_DB"   // DB12
VERSION : 0.1
// stored: AutoNumber false, DBAccessibleFromOPCUA true, InstanceOfName K12_出口自动, InstanceOfType FB
"K12_出口自动"
BEGIN
END_DATA_BLOCK

DATA_BLOCK "K13_ST01上自动_DB"   // DB13
VERSION : 0.1
// stored: AutoNumber false, DBAccessibleFromOPCUA true, InstanceOfName K13_ST01上自动, InstanceOfType FB
"K13_ST01上自动"
BEGIN
END_DATA_BLOCK

DATA_BLOCK "K14_ST02上自动_DB"   // DB14
VERSION : 0.1
// stored: AutoNumber false, DBAccessibleFromOPCUA true, InstanceOfName K14_ST02上自动, InstanceOfType FB
"K14_ST02上自动"
BEGIN
END_DATA_BLOCK

DATA_BLOCK "K15_ST03上自动_DB"   // DB15
VERSION : 0.1
// stored: AutoNumber false, DBAccessibleFromOPCUA true, InstanceOfName K15_ST03上自动, InstanceOfType FB
"K15_ST03上自动"
BEGIN
END_DATA_BLOCK

DATA_BLOCK "K16_ST04上自动_DB"   // DB16
VERSION : 0.1
// stored: AutoNumber false, DBAccessibleFromOPCUA true, InstanceOfName K16_ST04上自动, InstanceOfType FB
"K16_ST04上自动"
BEGIN
END_DATA_BLOCK

DATA_BLOCK "K17_ST05上自动_DB"   // DB17
VERSION : 0.1
// stored: AutoNumber false, DBAccessibleFromOPCUA true, InstanceOfName K17_ST05上自动, InstanceOfType FB
"K17_ST05上自动"
BEGIN
END_DATA_BLOCK

DATA_BLOCK "K18_ST06上自动_DB"   // DB18
VERSION : 0.1
// stored: AutoNumber false, DBAccessibleFromOPCUA true, InstanceOfName K18_ST06上自动, InstanceOfType FB
"K18_ST06上自动"
BEGIN
END_DATA_BLOCK

DATA_BLOCK "K19_ST07上自动_DB"   // DB19
VERSION : 0.1
// stored: AutoNumber false, DBAccessibleFromOPCUA true, InstanceOfName K19_ST07上自动, InstanceOfType FB
"K19_ST07上自动"
BEGIN
END_DATA_BLOCK

DATA_BLOCK "K20_ST08上自动_DB"   // DB20
VERSION : 0.1
// stored: AutoNumber false, DBAccessibleFromOPCUA true, InstanceOfName K20_ST08上自动, InstanceOfType FB
"K20_ST08上自动"
BEGIN
END_DATA_BLOCK

DATA_BLOCK "K21_ST09上自动_DB"   // DB21
VERSION : 0.1
// stored: AutoNumber false, DBAccessibleFromOPCUA true, InstanceOfName K21_ST09上自动, InstanceOfType FB
"K21_ST09上自动"
BEGIN
END_DATA_BLOCK

DATA_BLOCK "K22_ST10上自动_DB"   // DB22
VERSION : 0.1
// stored: AutoNumber false, DBAccessibleFromOPCUA true, InstanceOfName K22_ST10上自动, InstanceOfType FB
"K22_ST10上自动"
BEGIN
END_DATA_BLOCK

DATA_BLOCK "K23_ST11上自动_DB"   // DB23
VERSION : 0.1
// stored: AutoNumber false, DBAccessibleFromOPCUA true, InstanceOfName K23_ST11上自动, InstanceOfType FB
"K23_ST11上自动"
BEGIN
END_DATA_BLOCK

DATA_BLOCK "K24_ST12上自动_DB"   // DB24
VERSION : 0.1
// stored: AutoNumber false, DBAccessibleFromOPCUA true, InstanceOfName K24_ST12上自动, InstanceOfType FB
"K24_ST12上自动"
BEGIN
END_DATA_BLOCK

DATA_BLOCK "K25_ST03下自动_DB"   // DB25
VERSION : 0.1
// stored: AutoNumber false, DBAccessibleFromOPCUA true, InstanceOfName K25_ST03下自动, InstanceOfType FB
"K25_ST03下自动"
BEGIN
END_DATA_BLOCK

DATA_BLOCK "K26_ST02下自动_DB"   // DB26
VERSION : 0.1
// stored: AutoNumber false, DBAccessibleFromOPCUA true, InstanceOfName K26_ST02下自动, InstanceOfType FB
"K26_ST02下自动"
BEGIN
END_DATA_BLOCK

DATA_BLOCK "K27_ST01下自动_DB"   // DB27
VERSION : 0.1
// stored: AutoNumber false, DBAccessibleFromOPCUA true, InstanceOfName K27_ST01下自动, InstanceOfType FB
"K27_ST01下自动"
BEGIN
END_DATA_BLOCK

DATA_BLOCK "K40_互锁_DB"   // DB40
VERSION : 0.1
// stored: AutoNumber false, DBAccessibleFromOPCUA true, InstanceOfName K40_互锁, InstanceOfType FB
"K40_互锁"
BEGIN
END_DATA_BLOCK

DATA_BLOCK "SinaParaS_DB"   // DB303
// stored: AutoNumber false, DBAccessibleFromOPCUA true, InstanceOfName SinaParaS, OfSystemLibElement SinaParaS, OfSystemLibVersion 1.0
"SinaParaS"
   // VAR_INPUT
   //    Start : Bool;
   //    ReadWrite : Bool;
   //    Parameter : Int;
   //    Index : Int;
   //    ValueWrite1 : Real;
   //    ValueWrite2 : DInt;
   //    AxisNo : Byte;
   //    hardwareId : HW_IO;
   // END_VAR
   // VAR_OUTPUT
   //    Ready : Bool;
   //    Busy : Bool;
   //    Done : Bool;
   //    ValueRead1 : Real;
   //    ValueRead2 : DInt;
   //    Format : Byte;
   //    ErrorNo : Word;
   //    Error : Bool;
   //    ErrorId : DWord;
   //    DiagId : Word;
   // END_VAR
   // VAR
   //    sbWrError : Bool;
   //    sbWrDone : Bool;
   //    sbRdError : Bool;
   //    sbWrBusy : Bool;
   //    sbRdBusy : Bool;
   //    sbWrStart : Bool;
   //    sbRdStart : Bool;
   //    sbWrStart1 : Bool;
   //    sbRdStart1 : Bool;
   //    sbWrStart2 : Bool;
   //    sbRdStart2 : Bool;
   //    sbStart : Bool;
   //    sbReady : Bool;
   //    sbRead : Bool;
   //    sbWrite : Bool;
   //    sbParaNo : Bool;
   //    sbBusy : Bool;
   //    sbError : Bool;
   //    sbDone : Bool;
   //    syFormat : Byte;
   //    syAxisNo : Byte;
   //    siReqRef : Int;
   //    siErrorId : Int;
   //    siErrorCount : Int;
   //    siMaxErrCount : Int;
   //    swParaError : Word;
   //    sReqParaMulti { S7_SetPoint := 'True'} : SinaReqPara;
   //    sChaParaMulti { S7_SetPoint := 'True'} : SinaChaPara;
   //    sRespParaMulti { S7_SetPoint := 'True'} : SinaRespPara;
   //    RDREC_1 { S7_SetPoint := 'True'} : RDREC;
   //    WRREC_1 { S7_SetPoint := 'True'} : WRREC;
   //    siLenHeader : Int;
   //    siLenParaMulti : Int;
   //    siLenChaPara : Int;
   // END_VAR
BEGIN
END_DATA_BLOCK

DATA_BLOCK "SinaPosSer"   // DB300
// stored: AutoNumber false, DBAccessibleFromOPCUA true, InstanceOfName SinaPos, OfSystemLibElement SinaPos, OfSystemLibVersion 2.1
"SinaPos"
   // VAR_INPUT
   //    ModePos : Int;
   //    EnableAxis : Bool;
   //    CancelTraversing : Bool;
   //    IntermediateStop : Bool;
   //    Positive : Bool;
   //    Negative : Bool;
   //    Jog1 : Bool;
   //    Jog2 : Bool;
   //    FlyRef : Bool;
   //    AckError : Bool;
   //    ExecuteMode : Bool;
   //    Position : DInt;
   //    Velocity : DInt;
   //    OverV : Int;
   //    OverAcc : Int;
   //    OverDec : Int;
   //    ConfigEPos : DWord;
   //    HWIDSTW : HW_IO;
   //    HWIDZSW : HW_IO;
   // END_VAR
   // VAR_OUTPUT
   //    AxisEnabled : Bool;
   //    AxisPosOk : Bool;
   //    AxisSpFixed : Bool;
   //    AxisRef : Bool;
   //    AxisWarn : Bool;
   //    AxisError : Bool;
   //    Lockout : Bool;
   //    ActVelocity : DInt;
   //    ActPosition : DInt;
   //    ActMode : Int;
   //    EPosZSW1 : Word;
   //    EPosZSW2 : Word;
   //    ActWarn : Word;
   //    ActFault : Word;
   //    Error : Bool;
   //    Status : Word;
   //    DiagID : Word;
   // END_VAR
   // VAR
   //    sbOff1Edge : Bool;
   //    sbOff1 : Bool;
   //    sbExecuteEdge : Bool;
   //    sbExecute : Bool;
   //    sbRefTypEdge : Bool;
   //    sbRefTyp : Bool;
   //    sbMdiStart : Bool;
   //    sbMdiStartEdge : Bool;
   //    sbRefStart : Bool;
   //    sbJogInc : Bool;
   //    sbReady : Bool;
   //    sbIOp : Bool;
   //    sbAccel : Bool;
   //    sbDecel : Bool;
   //    sbAlarm : Bool;
   //    sbFault : Bool;
   //    sbFWD : Bool;
   //    sbBWD : Bool;
   //    sbBusy : Bool;
   //    swStatus : Word;
   //    swEPosZSW1 : Word;
   //    swEPosZSW2 : Word;
   //    siExecuteCyc : Int;
   //    siRefTypCyc : Int;
   //    siJogIncCyc : Int;
   //    siMdiStartCyc : Int;
   //    siRefActRetry : Int;
   //    siModePos : Int;
   //    siModePosMax : Int;
   //    siCycWait : Int;
   //    siRetryMax : Int;
   //    sbModePos : Bool;
   //    STW1 : Word;
   //    EPosSTW1 : Word;
   //    EPosSTW2 : Word;
   //    STW2 : Word;
   //    OverrideV : Word;
   //    PositionSP : DWord;
   //    VelocitySP : DWord;
   //    OverrideA : Word;
   //    OverrideD : Word;
   //    Reserve : Word;
   //    ZSW1 : Word;
   //    EPosZSW3 : Word;
   //    EPosZSW4 : Word;
   //    ZSW2 : Word;
   //    NotUsed : Word;
   //    PositionAV : DWord;
   //    VelocityAV : DWord;
   //    ErrNr : Word;
   //    WarnNr : Word;
   //    Reserve_1 : Word;
   // END_VAR
BEGIN
END_DATA_BLOCK
